(* IEC 61131-3 sources: SmartHomeNew/snapshots/2026-05-19 (part 3) *)

(* ---- FB_Heating_Runtime_Timeline_Observer.st ---- *)
// ==============================================================================
// Heating runtime timeline observer
// Read-only deterministic execution timeline layer.
// ==============================================================================
FUNCTION_BLOCK FB_Heating_Runtime_Timeline_Observer
VAR_INPUT
    VI_Enable : BOOL;
    VI_Frame : ST_Heating_Runtime_Execution_Frame;
END_VAR
VAR_IN_OUT
    VIO_Timeline : ST_Heating_Runtime_Execution_Timeline;
END_VAR
VAR
    L_Index : UINT;
END_VAR

IF NOT VI_Enable THEN
    RETURN;
END_IF;

// ======================================================
// SAFE INDEX NORMALIZATION
// ======================================================
IF (VIO_Timeline.Write_Index < 1) OR
   (VIO_Timeline.Write_Index >= 64) THEN

    L_Index := 1;

    IF VIO_Timeline.Write_Index >= 64 THEN
        VIO_Timeline.Timeline_Overflow := TRUE;
    END_IF;

ELSE
    L_Index := VIO_Timeline.Write_Index + 1;
END_IF;

// ======================================================
// FRAME STORAGE
// ======================================================
VIO_Timeline.Frames[L_Index] := VI_Frame;
VIO_Timeline.Write_Index := L_Index;

IF VIO_Timeline.Frame_Count < 64 THEN
    VIO_Timeline.Frame_Count :=
        VIO_Timeline.Frame_Count + 1;
END_IF;

// ======================================================
// TELEMETRY UPDATE
// ======================================================
VIO_Timeline.Sequencing_Valid :=
    VI_Frame.Sequencing_Valid;

VIO_Timeline.Ownership_Valid :=
    VI_Frame.Ownership_Valid;

VIO_Timeline.Synchronization_Valid :=
    VI_Frame.Synchronization_Valid;

VIO_Timeline.Runtime_Jitter_Detected :=
    VI_Frame.Runtime_Jitter_Detected;

VIO_Timeline.Runtime_Latency_Detected :=
    VI_Frame.Runtime_Latency_Detected;

VIO_Timeline.Runtime_Degraded :=
    VI_Frame.Runtime_Degraded;

VIO_Timeline.Status_Code := VI_Frame.Status_Code;
VIO_Timeline.Status_Text := VI_Frame.Status_Text;

END_FUNCTION_BLOCK
// >>> BULK_SYNC_ANCHOR: FB_Heating_Runtime_Timeline_Observer <<<

(* ---- FB_Heating_Safe_State.st ---- *)
FUNCTION_BLOCK FB_Heating_Safe_State
VAR_INPUT
    VI_Block_Normal_Heating : BOOL;
    VI_IO_Failsafe_Active : BOOL;
    VI_Gas_Safety_Active : BOOL;
    VI_Freeze_Active : BOOL;
    VI_Freeze_Target_Supply : REAL;
    VI_Manifold_Temps_Supply : ARRAY[1..GVL_CONSTANTS.C_MAX_MANIFOLDS] OF REAL;
    VI_Boiler_Error_Status : ARRAY[1..GVL_CONSTANTS.C_MAX_BOILERS] OF BOOL;
    VI_Boiler_OT_Online : ARRAY[1..GVL_CONSTANTS.C_MAX_BOILERS] OF BOOL;
END_VAR
VAR_OUTPUT
    VO_Applied : BOOL;
    VO_Zone_Valves : ARRAY[1..GVL_CONSTANTS.C_MAX_HEATING_CIRCUITS] OF BOOL;
    VO_Manifold_Pumps : ARRAY[1..GVL_CONSTANTS.C_MAX_MANIFOLDS] OF BOOL;
    VO_Manifold_Valves : ARRAY[1..GVL_CONSTANTS.C_MAX_MANIFOLDS] OF REAL;
    VO_Boiler_OT_Enable : ARRAY[1..GVL_CONSTANTS.C_MAX_BOILERS] OF BOOL;
    VO_Boiler_OT_Setpoint : ARRAY[1..GVL_CONSTANTS.C_MAX_BOILERS] OF REAL;
    VO_Boiler_Status : ARRAY[1..GVL_CONSTANTS.C_MAX_BOILERS] OF ST_Boiler_Status;
    VO_Backup_Circulation_Pump : BOOL;
    VO_Electric_Heater_Enable : BOOL;
    VO_Freeze_Risk_Status : BOOL;
END_VAR
VAR
    L_i : INT;
    L_Min_Supply_Temp : REAL;
    L_Freeze_Circulation_Required : BOOL;
END_VAR

VO_Applied := VI_Block_Normal_Heating;
VO_Backup_Circulation_Pump := FALSE;
VO_Electric_Heater_Enable := FALSE;
VO_Freeze_Risk_Status := FALSE;

L_Freeze_Circulation_Required := VI_Freeze_Active AND (VI_IO_Failsafe_Active OR VI_Gas_Safety_Active);

IF NOT VI_Block_Normal_Heating THEN
    RETURN;
END_IF;

// =============================
// ZONE VALVES (FIXED)
// =============================
FOR L_i := 1 TO GVL_CONSTANTS.C_MAX_HEATING_CIRCUITS DO
    IF L_Freeze_Circulation_Required THEN
        VO_Zone_Valves[L_i] := TRUE;
    ELSE
        VO_Zone_Valves[L_i] := FALSE;
    END_IF;
END_FOR;

// =============================
// MANIFOLD CONTROL
// =============================
FOR L_i := 1 TO GVL_CONSTANTS.C_MAX_MANIFOLDS DO
    IF L_Freeze_Circulation_Required THEN
        VO_Manifold_Pumps[L_i] := TRUE;
        VO_Manifold_Valves[L_i] := REAL#35.0;
    ELSE
        VO_Manifold_Pumps[L_i] := FALSE;
        VO_Manifold_Valves[L_i] := REAL#0.0;
    END_IF;
END_FOR;

// =============================
// BOILERS OFF
// =============================
FOR L_i := 1 TO GVL_CONSTANTS.C_MAX_BOILERS DO
    VO_Boiler_OT_Enable[L_i] := FALSE;
    VO_Boiler_OT_Setpoint[L_i] := REAL#0.0;
    VO_Boiler_Status[L_i].Warning := FALSE;
    VO_Boiler_Status[L_i].Error := TRUE;
END_FOR;

// =============================
// FREEZE PROTECTION LOGIC
// =============================
IF VI_Gas_Safety_Active AND VI_Freeze_Active THEN
    VO_Backup_Circulation_Pump := TRUE;

    L_Min_Supply_Temp := REAL#1000.0;
    FOR L_i := 1 TO GVL_CONSTANTS.C_MAX_MANIFOLDS DO
        IF VI_Manifold_Temps_Supply[L_i] < L_Min_Supply_Temp THEN
            L_Min_Supply_Temp := VI_Manifold_Temps_Supply[L_i];
        END_IF;
    END_FOR;

    IF L_Min_Supply_Temp > REAL#900.0 THEN
        L_Min_Supply_Temp := REAL#0.0;
    END_IF;

    IF L_Min_Supply_Temp < (VI_Freeze_Target_Supply - REAL#1.0) THEN
        VO_Electric_Heater_Enable := TRUE;
    ELSIF L_Min_Supply_Temp > (VI_Freeze_Target_Supply + REAL#1.0) THEN
        VO_Electric_Heater_Enable := FALSE;
    END_IF;

    VO_Freeze_Risk_Status := TRUE;
END_IF;

// =============================
// IO FAILSAFE + FREEZE
// =============================
IF VI_IO_Failsafe_Active AND VI_Freeze_Active THEN
    IF VI_Boiler_OT_Online[1] AND NOT VI_Boiler_Error_Status[1] THEN
        VO_Boiler_OT_Enable[1] := TRUE;
        VO_Boiler_OT_Setpoint[1] := VI_Freeze_Target_Supply;
    END_IF;
END_IF;

END_FUNCTION_BLOCK
// >>> BULK_SYNC_ANCHOR: FB_Heating_Safe_State <<<

(* ---- FB_Heating_System_Manager.st ---- *)
FUNCTION_BLOCK FB_Heating_System_Manager
VAR_INPUT
    VI_System_Mode : E_System_Operating_Mode;
    VI_System_Time_MS : UDINT;
    VI_IsActivePLC : BOOL;
    VI_Outdoor_Temp : REAL;
    VI_Config : ST_Heating_Config;
    VI_Tariff : ST_Tariff_Config;
    VI_Current_Hour : UINT;
    VI_DHW_Heating_Demand : BOOL;
    VI_DHW_Target_Temp : REAL;
    VI_Emergency_Stop : BOOL;
    VI_Gas_Safety_Stop : BOOL;
    VI_Boiler_Error_Status : ARRAY[1..GVL_CONSTANTS.C_MAX_BOILERS] OF BOOL;
    VI_Boiler_OT_Online : ARRAY[1..GVL_CONSTANTS.C_MAX_BOILERS] OF BOOL;
    VI_Boiler_Modulation : ARRAY[1..GVL_CONSTANTS.C_MAX_BOILERS] OF REAL;
END_VAR
VAR_IN_OUT
    VI_Floor_Temps : ARRAY[1..GVL_CONSTANTS.C_MAX_HEATING_CIRCUITS] OF REAL;
    VI_Room_Temps : ARRAY[1..GVL_CONSTANTS.C_MAX_ZONES] OF REAL;
    VI_Manifold_Pressures : ARRAY[1..GVL_CONSTANTS.C_MAX_MANIFOLDS] OF REAL;
    VI_Manifold_Currents : ARRAY[1..GVL_CONSTANTS.C_MAX_MANIFOLDS] OF REAL;
    VI_Manifold_Temps_Supply : ARRAY[1..GVL_CONSTANTS.C_MAX_MANIFOLDS] OF REAL;
    VI_Manifold_Temps_Return : ARRAY[1..GVL_CONSTANTS.C_MAX_MANIFOLDS] OF REAL;
    VI_Boiler_Flame_Status : ARRAY[1..GVL_CONSTANTS.C_MAX_BOILERS] OF BOOL;
    VI_Zone_Configs : ARRAY[1..GVL_CONSTANTS.C_MAX_HEATING_CIRCUITS] OF ST_FloorHeating_Circuit_Config;
    VI_Rule_Actions : ARRAY[1..GVL_CONSTANTS.C_MAX_RULES] OF ST_Rule_Action;
    VI_IO_Modules_Online : ARRAY[1..GVL_CONSTANTS.C_MAX_MODULES] OF BOOL;
    VI_Manifold_End_Switches : ARRAY[1..GVL_CONSTANTS.C_MAX_MANIFOLDS] OF BOOL;
    VI_Valve_Test_Config : ARRAY[1..GVL_CONSTANTS.C_MAX_MANIFOLDS] OF ST_Valve_Test_Config;
END_VAR
VAR_OUTPUT
    VO_Manifold_Valves : ARRAY[1..GVL_CONSTANTS.C_MAX_MANIFOLDS] OF REAL;
    VO_Manifold_Pumps : ARRAY[1..GVL_CONSTANTS.C_MAX_MANIFOLDS] OF BOOL;
    VO_Zone_Valves : ARRAY[1..GVL_CONSTANTS.C_MAX_HEATING_CIRCUITS] OF BOOL;
    VO_Boiler_OT_Enable : ARRAY[1..GVL_CONSTANTS.C_MAX_BOILERS] OF BOOL;
    VO_Boiler_OT_Setpoint : ARRAY[1..GVL_CONSTANTS.C_MAX_BOILERS] OF REAL;
    VO_Backup_Circulation_Pump : BOOL;
    VO_Electric_Heater_Enable : BOOL;
    VO_Freeze_Risk_Status : BOOL;
    VO_Status : ARRAY[1..GVL_CONSTANTS.C_MAX_MANIFOLDS] OF ST_Manifold_Status;
    VO_Boiler_Status : ARRAY[1..GVL_CONSTANTS.C_MAX_BOILERS] OF ST_Boiler_Status;
END_VAR
VAR
    L_i : INT;
    L_Target_Supply_Temp : REAL;
    L_Manifold_Demand_Map : ARRAY[1..GVL_CONSTANTS.C_MAX_MANIFOLDS] OF BOOL;
    L_Manifold_Demand_Filtered : ARRAY[1..GVL_CONSTANTS.C_MAX_MANIFOLDS] OF BOOL;
    L_Manifold_Available : ARRAY[1..GVL_CONSTANTS.C_MAX_MANIFOLDS] OF BOOL;
    L_Manifold_In_Service : ARRAY[1..GVL_CONSTANTS.C_MAX_MANIFOLDS] OF BOOL;
    L_Manifold_Subsystem_Degraded : ARRAY[1..GVL_CONSTANTS.C_MAX_MANIFOLDS] OF BOOL;
    L_Manifold_Base_Priority : ARRAY[1..GVL_CONSTANTS.C_MAX_MANIFOLDS] OF INT;
    L_Manifold_Effective_Priority : ARRAY[1..GVL_CONSTANTS.C_MAX_MANIFOLDS] OF INT;
    L_Manifold_Thermal_Weight : ARRAY[1..GVL_CONSTANTS.C_MAX_MANIFOLDS] OF REAL;
    L_Allocation_Degraded : BOOL;
    fbValveTestManager : FB_Valve_Test_Manager;
    L_IO_Failsafe_Active : BOOL;
    L_Freeze_Active : BOOL;
    L_Freeze_Target_Supply : REAL;
    L_Policy_Degraded : BOOL;
    L_Sensor_Error : BOOL;
    L_Subsys_Degraded : BOOL;
    L_Pressure_OK : BOOL;
    L_Prev_Pressure : ARRAY[1..GVL_CONSTANTS.C_MAX_MANIFOLDS] OF REAL;
    L_Prev_Current : ARRAY[1..GVL_CONSTANTS.C_MAX_MANIFOLDS] OF REAL;
    L_Confidence : REAL;
    L_Policy_Target_Adjustment : REAL;
    fbAdaptiveTarget : FB_Heating_Adaptive_Target;
    fbSafetyGate : FB_Heating_Safety_Gate;
    fbSafeState : FB_Heating_Safe_State;
    fbDemandMap : FB_Heating_Demand_Map;
    fbPolicyPriorityBridge : FB_Heating_Policy_Priority_Bridge;
    fbAllocationFilter : FB_Heating_Allocation_Filter;
    fbRuntimeObservability : FB_Heating_Runtime_Observability;
    fbCircuitControl : FB_Heating_Circuit_Control;
    fbManifoldControl : FB_Heating_Manifold_Control;
    fbBoilerControl : FB_Heating_Boiler_Control;
END_VAR

L_Policy_Degraded := (VI_System_Mode = E_System_Operating_Mode.MODE_DEGRADED);

GVL_STATE.G_Heating_IO_Fault := FALSE;
GVL_STATE.G_Heating_Sensor_Fault := FALSE;
GVL_STATE.G_Heating_Subsystem_Degraded := FALSE;
L_Sensor_Error := FALSE;
L_Subsys_Degraded := FALSE;
L_Allocation_Degraded := FALSE;

L_IO_Failsafe_Active := FALSE;
FOR L_i := 1 TO GVL_CONSTANTS.C_MAX_MODULES DO
    IF NOT VI_IO_Modules_Online[L_i] THEN
        L_IO_Failsafe_Active := TRUE;
        GVL_STATE.G_Heating_IO_Fault := TRUE;
        GVL_STATE.G_Heating_Subsystem_Degraded := TRUE;
        EXIT;
    END_IF;
END_FOR;

fbSafetyGate(
    VI_System_Mode := VI_System_Mode,
    VI_Emergency_Stop := VI_Emergency_Stop,
    VI_Gas_Safety_Stop := VI_Gas_Safety_Stop,
    VI_IO_Failsafe_Active := L_IO_Failsafe_Active,
    VI_Outdoor_Temp := VI_Outdoor_Temp,
    VI_Freeze_Threshold := VI_Config.Freeze_Threshold,
    VI_Floor_Temps := VI_Floor_Temps,
    VO_Freeze_Mode_Active => L_Freeze_Active,
    VO_Freeze_Target_Supply => L_Freeze_Target_Supply
);

fbSafeState(
    VI_Block_Normal_Heating := fbSafetyGate.VO_Block_Normal_Heating,
    VI_IO_Failsafe_Active := fbSafetyGate.VO_IO_Failsafe_Active,
    VI_Gas_Safety_Active := fbSafetyGate.VO_Gas_Safety_Active,
    VI_Freeze_Active := L_Freeze_Active,
    VI_Freeze_Target_Supply := L_Freeze_Target_Supply,
    VI_Manifold_Temps_Supply := VI_Manifold_Temps_Supply,
    VI_Boiler_Error_Status := VI_Boiler_Error_Status,
    VI_Boiler_OT_Online := VI_Boiler_OT_Online
);

IF fbSafeState.VO_Applied THEN
    FOR L_i := 1 TO GVL_CONSTANTS.C_MAX_HEATING_CIRCUITS DO
        VO_Zone_Valves[L_i] := fbSafeState.VO_Zone_Valves[L_i];
    END_FOR;

    FOR L_i := 1 TO GVL_CONSTANTS.C_MAX_MANIFOLDS DO
        VO_Manifold_Pumps[L_i] := fbSafeState.VO_Manifold_Pumps[L_i];
        VO_Manifold_Valves[L_i] := fbSafeState.VO_Manifold_Valves[L_i];
    END_FOR;

    FOR L_i := 1 TO GVL_CONSTANTS.C_MAX_BOILERS DO
        VO_Boiler_OT_Enable[L_i] := fbSafeState.VO_Boiler_OT_Enable[L_i];
        VO_Boiler_OT_Setpoint[L_i] := fbSafeState.VO_Boiler_OT_Setpoint[L_i];
        VO_Boiler_Status[L_i] := fbSafeState.VO_Boiler_Status[L_i];
    END_FOR;

    VO_Backup_Circulation_Pump := fbSafeState.VO_Backup_Circulation_Pump;
    VO_Electric_Heater_Enable := fbSafeState.VO_Electric_Heater_Enable;
    VO_Freeze_Risk_Status := fbSafeState.VO_Freeze_Risk_Status;
    RETURN;
END_IF;

VO_Backup_Circulation_Pump := FALSE;
VO_Electric_Heater_Enable := FALSE;
VO_Freeze_Risk_Status := FALSE;

IF L_Freeze_Active THEN
    L_Target_Supply_Temp := L_Freeze_Target_Supply;
ELSE
    L_Target_Supply_Temp := VI_Config.Target_Floor_Temp;
END_IF;

fbAdaptiveTarget(
    VI_Base_Target_Supply_Temp := L_Target_Supply_Temp,
    VI_Global_Target_Temperature := GVL_STATE.G_Target_Temperature,
    VI_Zone_Configs := VI_Zone_Configs,
    VI_Floor_Temps := VI_Floor_Temps,
    VI_Room_Temps := VI_Room_Temps,
    VO_Target_Supply_Temp => L_Target_Supply_Temp
);

L_Policy_Target_Adjustment := GVL_HEATING_POLICY.G_Policy_Target_Adjustment;

IF L_Policy_Target_Adjustment > REAL#5.0 THEN
    L_Policy_Target_Adjustment := REAL#5.0;
ELSIF L_Policy_Target_Adjustment < REAL#-3.0 THEN
    L_Policy_Target_Adjustment := REAL#-3.0;
END_IF;

L_Target_Supply_Temp :=
    LIMIT(
        GVL_CONSTANTS.C_BOILER_SETPOINT_MIN,
        L_Target_Supply_Temp + L_Policy_Target_Adjustment,
        GVL_CONSTANTS.C_BOILER_SETPOINT_MAX
    );

fbCircuitControl(
    VI_System_Time_MS := VI_System_Time_MS,
    VI_Current_Hour := VI_Current_Hour,
    VI_IsActivePLC := VI_IsActivePLC,
    VI_Config := VI_Config,
    VI_Tariff := VI_Tariff,
    VI_Scenario_Adjust := REAL#0.0,
    VI_Zone_Configs := VI_Zone_Configs,
    VI_Floor_Temps := VI_Floor_Temps,
    VI_Room_Temps := VI_Room_Temps,
    VI_Rule_Actions := VI_Rule_Actions,
    VO_Zone_Valves => VO_Zone_Valves,
    VO_Heating_Sensor_Fault => L_Sensor_Error
);

GVL_STATE.G_Heating_Sensor_Fault := L_Sensor_Error;

fbDemandMap(
    VI_Zone_Valves := VO_Zone_Valves,
    VI_Zone_Configs := VI_Zone_Configs,
    VO_Manifold_Demand_Map => L_Manifold_Demand_Map
);

FOR L_i := 1 TO GVL_CONSTANTS.C_MAX_MANIFOLDS DO
    L_Manifold_Available[L_i] := VI_Manifold_Pressures[L_i] >= GVL_CONSTANTS.C_MIN_HEATING_MANIFOLD_PRESSURE;
    L_Manifold_In_Service[L_i] := GVL_CONFIG.G_Manifold_Pump_In_Service[L_i];
    L_Manifold_Subsystem_Degraded[L_i] :=
        GVL_STATE.G_Predictive_Pump_Pressure_Drop[L_i]
        OR GVL_STATE.G_Predictive_Pump_Current_Rise[L_i];

    L_Manifold_Base_Priority[L_i] := GVL_CONFIG.G_Manifold_Priority[L_i];
    L_Manifold_Thermal_Weight[L_i] := GVL_CONFIG.G_Manifold_Thermal_Weight[L_i];
END_FOR;

fbPolicyPriorityBridge(
    VI_Enable := (GVL_CONFIG.G_Max_Thermal_Budget > REAL#0.0),
    VI_Zone_Valves := VO_Zone_Valves,
    VI_Zone_Configs := VI_Zone_Configs,
    VI_Manifold_Base_Priority := L_Manifold_Base_Priority,
    VI_Zone_Priority_Bias := GVL_HEATING_POLICY.G_Zone_Priority_Bias,
    VI_Policy_Priority_Multiplier := GVL_HEATING_POLICY.G_Policy_Priority_Multiplier,
    VO_Manifold_Effective_Priority => L_Manifold_Effective_Priority
);

fbAllocationFilter(
    VI_Enable := TRUE,
    VI_Enable_Policy_Allocation := (GVL_CONFIG.G_Max_Thermal_Budget > REAL#0.0),
    VI_Freeze_Mode_Active := L_Freeze_Active,
    VI_DHW_Heating_Demand := VI_DHW_Heating_Demand,
    VI_Manifold_Demand_Map := L_Manifold_Demand_Map,
    VI_Manifold_Available := L_Manifold_Available,
    VI_Manifold_In_Service := L_Manifold_In_Service,
    VI_Manifold_Subsystem_Degraded := L_Manifold_Subsystem_Degraded,
    VI_Manifold_Base_Priority := L_Manifold_Effective_Priority,
    VI_Manifold_Thermal_Weight := L_Manifold_Thermal_Weight,
    VI_Max_Thermal_Budget := GVL_CONFIG.G_Max_Thermal_Budget,
    VO_Manifold_Demand_Filtered => L_Manifold_Demand_Filtered,
    VO_Allocation_Degraded => L_Allocation_Degraded
);

fbRuntimeObservability(
    VI_Policy_Active := (GVL_CONFIG.G_Max_Thermal_Budget > REAL#0.0),
    VI_Freeze_Bypass_Active := L_Freeze_Active,
    VI_DHW_Bypass_Active := VI_DHW_Heating_Demand,
    VI_Budget_Max := GVL_CONFIG.G_Max_Thermal_Budget,
    VI_Budget_Used := fbAllocationFilter.VO_Thermal_Budget_Used,
    VI_Requested := L_Manifold_Demand_Map,
    VI_Allowed := fbAllocationFilter.VO_Manifold_Allowed,
    VI_Filtered := L_Manifold_Demand_Filtered,
    VI_Block_Reason := fbAllocationFilter.VO_Manifold_Block_Reason,
    VI_Effective_Priority := fbAllocationFilter.VO_Manifold_Priority_Effective,
    VI_Priority_Bridge_Active := fbPolicyPriorityBridge.VO_Bridge_Active,
    VI_Priority_Bias_Applied := fbPolicyPriorityBridge.VO_Manifold_Priority_Bias_Applied,
    VI_Priority_Effective := L_Manifold_Effective_Priority
);

IF L_Allocation_Degraded THEN
    GVL_STATE.G_Heating_Subsystem_Degraded := TRUE;
END_IF;

fbManifoldControl(
    VI_System_Time_MS := VI_System_Time_MS,
    VI_IsActivePLC := VI_IsActivePLC,
    VI_DHW_Heating_Demand := VI_DHW_Heating_Demand,
    VI_Freeze_Mode_Active := L_Freeze_Active,
    VI_Target_Supply_Temp := L_Target_Supply_Temp,
    VI_Any_Zone_Active := L_Manifold_Demand_Filtered,
    VI_Manifold_Pressures := VI_Manifold_Pressures,
    VI_Manifold_Currents := VI_Manifold_Currents,
    VI_Manifold_Temps_Supply := VI_Manifold_Temps_Supply,
    VI_Manifold_Temps_Return := VI_Manifold_Temps_Return,
    VO_Manifold_Pumps => VO_Manifold_Pumps,
    VO_Manifold_Valves => VO_Manifold_Valves,
    VO_Status => VO_Status
);

FOR L_i := 1 TO GVL_CONSTANTS.C_MAX_MANIFOLDS DO
    L_Pressure_OK := VI_Manifold_Pressures[L_i] >= GVL_CONSTANTS.C_MIN_HEATING_MANIFOLD_PRESSURE;

    IF VO_Manifold_Pumps[L_i] AND NOT L_Pressure_OK THEN
        VO_Manifold_Pumps[L_i] := FALSE;
        GVL_STATE.G_Heating_Subsystem_Degraded := TRUE;
    END_IF;

    IF (L_Prev_Pressure[L_i] > REAL#0.0) AND ((L_Prev_Pressure[L_i] - VI_Manifold_Pressures[L_i]) > REAL#0.2) THEN
        GVL_STATE.G_Predictive_Pump_Pressure_Drop[L_i] := TRUE;
    ELSE
        GVL_STATE.G_Predictive_Pump_Pressure_Drop[L_i] := FALSE;
    END_IF;

    IF (L_Prev_Current[L_i] > REAL#0.0) AND (VI_Manifold_Currents[L_i] > (L_Prev_Current[L_i] * REAL#1.2)) THEN
        GVL_STATE.G_Predictive_Pump_Current_Rise[L_i] := TRUE;
    ELSE
        GVL_STATE.G_Predictive_Pump_Current_Rise[L_i] := FALSE;
    END_IF;

    IF GVL_STATE.G_Predictive_Pump_Pressure_Drop[L_i] OR GVL_STATE.G_Predictive_Pump_Current_Rise[L_i] THEN
        GVL_STATE.G_Heating_Subsystem_Degraded := TRUE;
    END_IF;

    L_Prev_Pressure[L_i] := VI_Manifold_Pressures[L_i];
    L_Prev_Current[L_i] := VI_Manifold_Currents[L_i];
END_FOR;

// ======================================================
// HEATING CONFIDENCE PUBLICATION
// ======================================================
// The former local error-score decay path has been replaced by the
// normalized input confidence surface. Runtime faults may still reduce
// confidence and reason publication, but the base confidence now comes
// from canonical input semantics.
L_Confidence := GVL_INPUT.IN_Min_Zone_Confidence;

IF L_Confidence < REAL#0.0 THEN
    L_Confidence := REAL#0.0;
ELSIF L_Confidence > REAL#1.0 THEN
    L_Confidence := REAL#1.0;
END_IF;

GVL_STATE.G_Heating_Confidence_Reason_Code := 0;
GVL_STATE.G_Heating_Confidence_Reason_Text := 'OK';

IF GVL_INPUT.IN_Input_Degraded OR GVL_INPUT.IN_Anomaly_Detected THEN
    GVL_STATE.G_Heating_Subsystem_Degraded := TRUE;
    GVL_STATE.G_Heating_Confidence_Reason_Code := 5;

    IF GVL_INPUT.IN_Anomaly_Reason <> '' THEN
        GVL_STATE.G_Heating_Confidence_Reason_Text := GVL_INPUT.IN_Anomaly_Reason;
    ELSE
        GVL_STATE.G_Heating_Confidence_Reason_Text := 'Input quality degraded';
    END_IF;
END_IF;

IF GVL_STATE.G_Heating_IO_Fault THEN
    IF L_Confidence > REAL#0.8 THEN
        L_Confidence := REAL#0.8;
    END_IF;
    GVL_STATE.G_Heating_Confidence_Reason_Code := 2;
    GVL_STATE.G_Heating_Confidence_Reason_Text := 'IO fault detected';
ELSIF GVL_STATE.G_Heating_Sensor_Fault THEN
    IF L_Confidence > REAL#0.6 THEN
        L_Confidence := REAL#0.6;
    END_IF;
    GVL_STATE.G_Heating_Confidence_Reason_Code := 1;
    GVL_STATE.G_Heating_Confidence_Reason_Text := 'Sensor fault detected';
ELSE
    FOR L_i := 1 TO GVL_CONSTANTS.C_MAX_MANIFOLDS DO
        IF VI_Manifold_Pressures[L_i] < GVL_CONSTANTS.C_MIN_HEATING_MANIFOLD_PRESSURE THEN
            IF L_Confidence > REAL#0.7 THEN
                L_Confidence := REAL#0.7;
            END_IF;
            GVL_STATE.G_Heating_Confidence_Reason_Code := 3;
            GVL_STATE.G_Heating_Confidence_Reason_Text := 'Low manifold pressure';
            EXIT;
        END_IF;
    END_FOR;

    FOR L_i := 1 TO GVL_CONSTANTS.C_MAX_MANIFOLDS DO
        IF GVL_STATE.G_Predictive_Pump_Pressure_Drop[L_i] OR GVL_STATE.G_Predictive_Pump_Current_Rise[L_i] THEN
            IF L_Confidence > REAL#0.75 THEN
                L_Confidence := REAL#0.75;
            END_IF;
            GVL_STATE.G_Heating_Confidence_Reason_Code := 4;
            GVL_STATE.G_Heating_Confidence_Reason_Text := 'Predictive pump degradation';
            EXIT;
        END_IF;
    END_FOR;
END_IF;

GVL_STATE.G_Heating_Confidence := L_Confidence;
GVL_STATE.G_Heating_Error_Score := REAL#1.0 - L_Confidence;

IF GVL_STATE.G_Heating_Confidence < REAL#0.5 THEN
    L_Target_Supply_Temp := L_Target_Supply_Temp - REAL#3.0;
END_IF;

CASE GVL_STATE.G_Heating_Confidence_Reason_Code OF
    1:
        L_Target_Supply_Temp := LIMIT(GVL_CONSTANTS.C_BOILER_SETPOINT_MIN, REAL#40.0, GVL_CONSTANTS.C_BOILER_SETPOINT_MAX);
    2:
        VO_Backup_Circulation_Pump := TRUE;
    3:
        FOR L_i := 1 TO GVL_CONSTANTS.C_MAX_MANIFOLDS DO
            VO_Manifold_Pumps[L_i] := FALSE;
        END_FOR;
    4:
        L_Target_Supply_Temp := LIMIT(GVL_CONSTANTS.C_BOILER_SETPOINT_MIN, L_Target_Supply_Temp - REAL#5.0, GVL_CONSTANTS.C_BOILER_SETPOINT_MAX);
    5:
        // Input-quality degradation is published for explainability first.
        // Runtime suppression remains governed by existing sensor validation
        // and safety/pressure ownership paths.
ELSE
    // no auto-recovery action
END_CASE;

fbValveTestManager(
    VI_System_Time_MS := VI_System_Time_MS,
    VI_IsActivePLC := VI_IsActivePLC,
    VI_Valve_Currents := VI_Manifold_Currents,
    VI_Valve_End_Switches := VI_Manifold_End_Switches,
    VI_Config := VI_Valve_Test_Config
);

IF fbValveTestManager.VO_Test_Active THEN
    L_i := fbValveTestManager.VO_Current_Valve;
    IF L_i >= 1 AND L_i <= GVL_CONSTANTS.C_MAX_MANIFOLDS THEN
        IF fbValveTestManager.VO_Valve_Cmd[L_i] THEN
            VO_Manifold_Valves[L_i] := REAL#100.0;
        ELSE
            VO_Manifold_Valves[L_i] := REAL#0.0;
        END_IF;
        VO_Manifold_Pumps[L_i] := FALSE;
    END_IF;
END_IF;

fbBoilerControl(
    VI_System_Time_MS := VI_System_Time_MS,
    VI_IsActivePLC := VI_IsActivePLC,
    VI_DHW_Heating_Demand := VI_DHW_Heating_Demand,
    VI_DHW_Target_Temp := VI_DHW_Target_Temp,
    VI_Target_Supply_Temp := L_Target_Supply_Temp,
    VI_Freeze_Mode_Active := L_Freeze_Active,
    VI_Policy_Degraded := L_Policy_Degraded,
    VI_Manifold_Pumps := VO_Manifold_Pumps,
    VI_Manifold_Valves := VO_Manifold_Valves,
    VI_Boiler_Flame_Status := VI_Boiler_Flame_Status,
    VI_Boiler_Error_Status := VI_Boiler_Error_Status,
    VI_Boiler_OT_Online := VI_Boiler_OT_Online,
    VI_Boiler_Modulation := VI_Boiler_Modulation,
    VO_Boiler_OT_Enable => VO_Boiler_OT_Enable,
    VO_Boiler_OT_Setpoint => VO_Boiler_OT_Setpoint,
    VO_Boiler_Status => VO_Boiler_Status,
    VO_Any_Subsystem_Degraded => L_Subsys_Degraded
);

GVL_STATE.G_Heating_Subsystem_Degraded := GVL_STATE.G_Heating_Subsystem_Degraded OR L_Subsys_Degraded;

END_FUNCTION_BLOCK
// >>> BULK_SYNC_ANCHOR: FB_Heating_System_Manager <<<

(* ---- FB_History_Manager.st ---- *)
FUNCTION_BLOCK FB_History_Manager
VAR_INPUT
    VI_System_Time_MS : UDINT;
    VI_Write_Event    : BOOL;
    VI_Event          : ST_History_Record;
END_VAR
VAR_OUTPUT
    VO_Total_Events   : UDINT;
END_VAR
VAR
    L_Prev_Write_Event : BOOL;
END_VAR

IF VI_Write_Event AND NOT L_Prev_Write_Event THEN
    GVL_Retain.G_History_Buffer[GVL_Retain.G_History_Write_Idx] := VI_Event;
    GVL_Retain.G_History_Buffer[GVL_Retain.G_History_Write_Idx].timestamp_ms := VI_System_Time_MS;

    GVL_Retain.G_History_Write_Idx := (GVL_Retain.G_History_Write_Idx MOD GVL_CONSTANTS.C_MAX_HISTORY_RECORDS) + 1;
    GVL_Retain.G_History_Total_Events := GVL_Retain.G_History_Total_Events + 1;
END_IF;
L_Prev_Write_Event := VI_Write_Event;

VO_Total_Events := GVL_Retain.G_History_Total_Events;
// >>> BULK_SYNC_ANCHOR: FB_History_Manager <<<
END_FUNCTION_BLOCK

(* ---- FB_HMI_Config_Workflow_Runtime.st ---- *)
FUNCTION_BLOCK FB_HMI_Config_Workflow_Runtime
VAR_INPUT
    VI_Enable : BOOL;
    VI_System_Time_MS : UDINT;
END_VAR
VAR
    L_State : ST_HMI_Config_Workflow_State;
END_VAR

IF NOT VI_Enable THEN
    GVL_HMI_Config_Workflow.G_Runtime_Valid := FALSE;
    RETURN;
END_IF;

L_State.Runtime_Valid := TRUE;
L_State.Runtime_System_Time_MS := VI_System_Time_MS;

L_State.Editor_Open :=
    GVL_HMI_Config_Workflow.G_Open_Editor_Request;

L_State.Validation_Requested :=
    GVL_HMI_Config_Workflow.G_Validate_Request;

L_State.Activation_Requested :=
    GVL_HMI_Config_Workflow.G_Activate_Request;

L_State.Rollback_Requested :=
    GVL_HMI_Config_Workflow.G_Rollback_Request;

L_State.Active_Version :=
    GVL_Water_Topology_Config.G_Active_Config_Version;

L_State.Draft_Version :=
    GVL_Config_Activation.G_Staged_Config_Version;

L_State.Last_Stable_Version :=
    GVL_Config_Activation.G_Last_Stable_Config_Version;

L_State.Quarantine_Visible :=
    GVL_Config_Activation.G_Config_Quarantine_Active;

L_State.Service_Mode_Required := TRUE;
L_State.Operator_Ack_Required := TRUE;

IF L_State.Editor_Open THEN
    L_State.Edit_Session_Active := TRUE;
END_IF;

IF L_State.Validation_Requested THEN

    IF GVL_Config_Activation.G_Activation_State.Staged_Config_Valid THEN

        L_State.Validation_OK := TRUE;

    ELSE

        L_State.Validation_Failed := TRUE;

    END_IF;

END_IF;

IF L_State.Activation_Requested THEN

    IF GVL_HMI_Config_Workflow.G_Service_Mode_Active
       AND GVL_HMI_Config_Workflow.G_Operator_Ack
       AND L_State.Validation_OK THEN

        L_State.Activation_Allowed := TRUE;
        GVL_Config_Activation.G_Activation_Request := TRUE;

    ELSE

        L_State.Activation_Blocked := TRUE;

    END_IF;

END_IF;

IF L_State.Rollback_Requested THEN

    IF GVL_HMI_Config_Workflow.G_Operator_Ack THEN

        L_State.Rollback_Allowed := TRUE;
        GVL_Config_Activation.G_Rollback_Request := TRUE;

    END_IF;

END_IF;

IF L_State.Activation_Blocked THEN

    L_State.Status_Code := 2;
    L_State.Status_Text := 'HMI activation blocked';

ELSIF L_State.Validation_Failed THEN

    L_State.Status_Code := 1;
    L_State.Status_Text := 'HMI validation failed';

ELSE

    L_State.Status_Code := 0;
    L_State.Status_Text := 'HMI config workflow healthy';

END_IF;

GVL_HMI_Config_Workflow.G_Workflow_State := L_State;

GVL_HMI_Config_Workflow.G_Runtime_Valid := TRUE;
GVL_HMI_Config_Workflow.G_Last_Update_MS := VI_System_Time_MS;
GVL_HMI_Config_Workflow.G_Status_Code := L_State.Status_Code;
GVL_HMI_Config_Workflow.G_Status_Text := L_State.Status_Text;

END_FUNCTION_BLOCK

(* ---- FB_IO_Module_Watchdog.st ---- *)
FUNCTION_BLOCK FB_IO_Module_Watchdog
VAR_INPUT
    VI_System_Time_MS : UDINT;
    VI_Module_ID : BYTE;
    VI_Heartbeat_Signal : BOOL; // Сигнал от модуля (например, мигающий бит)
    VI_Timeout_MS : UDINT := 2000; // Таймаут 2 секунды по умолчанию
END_VAR
VAR_OUTPUT
    VO_Module_Online : BOOL;
    VO_Error_Active : BOOL;
END_VAR
VAR
    L_Last_Heartbeat_State : BOOL;
    L_Last_Heartbeat_Time : UDINT;
    L_Elapsed_Time : UDINT;
END_VAR

// Отслеживание изменения сигнала
IF VI_Heartbeat_Signal <> L_Last_Heartbeat_State THEN
    L_Last_Heartbeat_Time := VI_System_Time_MS;
    L_Last_Heartbeat_State := VI_Heartbeat_Signal;
END_IF;

// Проверка таймаута
L_Elapsed_Time := (SEL(VI_System_Time_MS >= L_Last_Heartbeat_Time, VI_System_Time_MS - L_Last_Heartbeat_Time, (4294967295 - L_Last_Heartbeat_Time) + VI_System_Time_MS + 1));

IF L_Elapsed_Time > VI_Timeout_MS THEN
    VO_Module_Online := FALSE;
    VO_Error_Active := TRUE;
ELSE
    VO_Module_Online := TRUE;
    VO_Error_Active := FALSE;
END_IF;
// >>> BULK_SYNC_ANCHOR: FB_IO_Module_Watchdog <<<
END_FUNCTION_BLOCK

(* ---- FB_Lifetime_Predictor.st ---- *)
FUNCTION_BLOCK FB_Lifetime_Predictor
VAR_INPUT
    VI_Runtime_Hours : UDINT;
    VI_Start_Count   : UDINT;
    VI_Nominal_Life  : UDINT := 10000;
END_VAR
VAR_OUTPUT
    VO_Remaining_Percent : BYTE;
    VO_Maintenance_Req   : BOOL;
END_VAR

// Упрощенная модель износа
IF VI_Nominal_Life > 0 THEN
    VO_Remaining_Percent := TO_BYTE(100 - (VI_Runtime_Hours * 100 / VI_Nominal_Life));
ELSE
    VO_Remaining_Percent := 0;
END_IF;

VO_Maintenance_Req := (VO_Remaining_Percent < 10);
END_FUNCTION_BLOCK

(* ---- FB_Lighting_Blinds_Manager.st ---- *)
FUNCTION_BLOCK FB_Lighting_Blinds_Manager
VAR_INPUT
    VI_System_Time_MS : UDINT;
    VI_IsActivePLC : BOOL;
    VI_Current_Scenario : E_SCENARIO_TYPE;
    VI_Away_Level : BYTE;
    VI_Simulation_Active : BOOL;
    VI_Is_Night : BOOL;
    VI_System_Mode : E_System_Operating_Mode;
END_VAR
VAR_IN_OUT
    VI_Manual_Light_Override : ARRAY[1..GVL_CONSTANTS.C_MAX_LIGHT_ZONES] OF BYTE;
    VI_Manual_Blinds_Override : ARRAY[1..GVL_CONSTANTS.C_MAX_BLINDS] OF BYTE;
    VI_Simulation_Lights : ARRAY[1..GVL_CONSTANTS.C_MAX_LIGHT_ZONES] OF BOOL;
    VI_Physical_Switches : ARRAY[1..GVL_CONSTANTS.C_MAX_LIGHT_ZONES] OF BOOL;
    VI_Motion_Sensors : ARRAY[1..GVL_CONSTANTS.C_MAX_LIGHT_ZONES] OF BOOL;
    VI_Rule_Actions : ARRAY[1..GVL_CONSTANTS.C_MAX_RULES] OF ST_Rule_Action;
    VI_IO_Modules_Online : ARRAY[1..GVL_CONSTANTS.C_MAX_MODULES] OF BOOL;
    VI_Wet_Zone_Map : ARRAY[1..GVL_CONSTANTS.C_MAX_LIGHT_ZONES] OF BOOL;
    VI_Scenario_Configs : ARRAY[1..GVL_CONSTANTS.C_MAX_SCENARIOS] OF ST_Scenario_Config;
END_VAR
VAR_OUTPUT
    VO_Lighting_Levels : ARRAY[1..GVL_CONSTANTS.C_MAX_LIGHT_ZONES] OF BYTE;
    VO_Blinds_Positions : ARRAY[1..GVL_CONSTANTS.C_MAX_BLINDS] OF BYTE;
    VO_Wet_Zone_Light_Active : ARRAY[1..GVL_CONSTANTS.C_MAX_WET_ZONES] OF BOOL;
END_VAR
VAR
    L_i : INT;
    L_j : INT;
    L_Base_Light : BYTE;
    L_Base_Blinds : BYTE;
    L_Target_Base_Light : BYTE;
    L_Target_Base_Blinds : BYTE;
    L_Prev_Scenario : E_SCENARIO_TYPE;
    L_Transition_Light : FB_Scenario_Transition_Controller;
    L_Transition_Blinds : FB_Scenario_Transition_Controller;
    L_Light_States : ARRAY[1..GVL_CONSTANTS.C_MAX_LIGHT_ZONES] OF BOOL;
    L_Prev_Switches : ARRAY[1..GVL_CONSTANTS.C_MAX_LIGHT_ZONES] OF BOOL;
    L_Prev_Motion_Q : ARRAY[1..GVL_CONSTANTS.C_MAX_LIGHT_ZONES] OF BOOL;
    L_Manual_Override : ARRAY[1..GVL_CONSTANTS.C_MAX_LIGHT_ZONES] OF BOOL;
    L_Motion_Timers : ARRAY[1..GVL_CONSTANTS.C_MAX_LIGHT_ZONES] OF FB_System_Timer_TOF;
    L_Rule_Light_Active : BOOL;
    L_Rule_Light_Val : BYTE;
    L_Rule_Blinds_Active : BOOL;
    L_Rule_Blinds_Val : BYTE;
    L_Wet_Zone_Idx : INT;
    L_Effective_Scenario : E_SCENARIO_TYPE;
    L_Effective_Simulation_Active : BOOL;
END_VAR

IF NOT VI_IsActivePLC THEN RETURN; END_IF;

GVL_STATE.G_Lighting_IO_Fault := FALSE;
GVL_STATE.G_Lighting_Subsystem_Degraded := FALSE;

L_Effective_Scenario := VI_Current_Scenario;
L_Effective_Simulation_Active := VI_Simulation_Active;

CASE VI_System_Mode OF
    E_System_Operating_Mode.MODE_SAFE_STOP:
        FOR L_j := 1 TO GVL_CONSTANTS.C_MAX_LIGHT_ZONES DO
            VO_Lighting_Levels[L_j] := 0;
        END_FOR;
        FOR L_j := 1 TO GVL_CONSTANTS.C_MAX_BLINDS DO
            VO_Blinds_Positions[L_j] := 100;
        END_FOR;
        FOR L_j := 1 TO GVL_CONSTANTS.C_MAX_WET_ZONES DO
            VO_Wet_Zone_Light_Active[L_j] := FALSE;
        END_FOR;
        RETURN;
    E_System_Operating_Mode.MODE_FREEZE_PROTECTION:
        L_Effective_Scenario := E_SCENARIO_TYPE.SCENARIO_NONE;
        L_Effective_Simulation_Active := FALSE;
    E_System_Operating_Mode.MODE_DEGRADED:
        L_Effective_Simulation_Active := FALSE;
END_CASE;

L_Wet_Zone_Idx := 1;
FOR L_i := 1 TO GVL_CONSTANTS.C_MAX_WET_ZONES DO
    VO_Wet_Zone_Light_Active[L_i] := FALSE;
END_FOR;

FOR L_i := 1 TO GVL_CONSTANTS.C_MAX_MODULES DO
    IF NOT VI_IO_Modules_Online[L_i] THEN
        GVL_STATE.G_Lighting_IO_Fault := TRUE;
        GVL_STATE.G_Lighting_Subsystem_Degraded := TRUE;
        FOR L_j := 1 TO GVL_CONSTANTS.C_MAX_LIGHT_ZONES DO
            VO_Lighting_Levels[L_j] := 0;
        END_FOR;
        FOR L_j := 1 TO GVL_CONSTANTS.C_MAX_BLINDS DO
            VO_Blinds_Positions[L_j] := 100;
        END_FOR;
        RETURN;
    END_IF;
END_FOR;

IF L_Effective_Scenario >= 1 AND L_Effective_Scenario <= GVL_CONSTANTS.C_MAX_SCENARIOS THEN
    L_Target_Base_Light := VI_Scenario_Configs[L_Effective_Scenario].lighting_level_base;
    L_Target_Base_Blinds := VI_Scenario_Configs[L_Effective_Scenario].blinds_position_percent;
ELSE
    L_Target_Base_Light := 100;
    L_Target_Base_Blinds := 100;
END_IF;

IF VI_Is_Night AND L_Effective_Scenario <> E_SCENARIO_TYPE.SCENARIO_AWAY AND L_Effective_Scenario <> E_SCENARIO_TYPE.SCENARIO_SLEEP THEN
    L_Target_Base_Blinds := 0;
END_IF;

IF L_Effective_Scenario <> L_Prev_Scenario THEN
    L_Transition_Light(VI_System_Time := VI_System_Time_MS, VI_Start_Time := VI_System_Time_MS, VI_Duration := 5000, VI_Start_Value := TO_REAL(L_Base_Light), VI_End_Value := TO_REAL(L_Target_Base_Light));
    L_Transition_Blinds(VI_System_Time := VI_System_Time_MS, VI_Start_Time := VI_System_Time_MS, VI_Duration := 10000, VI_Start_Value := TO_REAL(L_Base_Blinds), VI_End_Value := TO_REAL(L_Target_Base_Blinds));
    L_Prev_Scenario := L_Effective_Scenario;
ELSE
    L_Transition_Light(VI_System_Time := VI_System_Time_MS, VI_Start_Time := L_Transition_Light.VI_Start_Time, VI_Duration := L_Transition_Light.VI_Duration, VI_Start_Value := L_Transition_Light.VI_Start_Value, VI_End_Value := TO_REAL(L_Target_Base_Light));
    L_Transition_Blinds(VI_System_Time := VI_System_Time_MS, VI_Start_Time := L_Transition_Blinds.VI_Start_Time, VI_Duration := L_Transition_Blinds.VI_Duration, VI_Start_Value := L_Transition_Blinds.VI_Start_Value, VI_End_Value := TO_REAL(L_Target_Base_Blinds));
END_IF;

L_Base_Light := TO_BYTE(L_Transition_Light.VO_Current_Value);
L_Base_Blinds := TO_BYTE(L_Transition_Blinds.VO_Current_Value);

FOR L_i := 1 TO GVL_CONSTANTS.C_MAX_LIGHT_ZONES DO
    L_Rule_Light_Active := FALSE;
    L_Rule_Light_Val := 0;
    FOR L_j := 1 TO GVL_CONSTANTS.C_MAX_RULES DO
        IF VI_Rule_Actions[L_j].Active AND VI_Rule_Actions[L_j].Target_ID = L_i THEN
            IF VI_Rule_Actions[L_j].Action_Type = E_Rule_Action_Type.ACTION_SET_LIGHTING_BASE THEN
                L_Rule_Light_Active := TRUE;
                L_Rule_Light_Val := REAL_TO_BYTE(VI_Rule_Actions[L_j].Value);
                L_Light_States[L_i] := (L_Rule_Light_Val > 0);
            ELSIF VI_Rule_Actions[L_j].Action_Type = E_Rule_Action_Type.ACTION_TOGGLE_LIGHTING AND VI_Rule_Actions[L_j].Triggered THEN
                L_Light_States[L_i] := NOT L_Light_States[L_i];
            END_IF;
        END_IF;
    END_FOR;

    IF VI_Physical_Switches[L_i] AND NOT L_Prev_Switches[L_i] THEN
        L_Light_States[L_i] := NOT L_Light_States[L_i];
        L_Manual_Override[L_i] := TRUE;
    END_IF;
    L_Prev_Switches[L_i] := VI_Physical_Switches[L_i];

    L_Motion_Timers[L_i](IN := VI_Motion_Sensors[L_i], PT := T#5m, VI_System_Time_MS := VI_System_Time_MS);

    IF L_Prev_Motion_Q[L_i] AND NOT L_Motion_Timers[L_i].Q THEN
        L_Manual_Override[L_i] := FALSE;
    END_IF;
    L_Prev_Motion_Q[L_i] := L_Motion_Timers[L_i].Q;

    IF L_Motion_Timers[L_i].Q THEN
        IF NOT L_Manual_Override[L_i] THEN
            L_Light_States[L_i] := TRUE;
        END_IF;
    ELSE
        IF NOT L_Manual_Override[L_i] THEN
            L_Light_States[L_i] := FALSE;
        END_IF;
    END_IF;

    IF L_Effective_Scenario = E_SCENARIO_TYPE.SCENARIO_AWAY AND L_Effective_Simulation_Active THEN
        L_Light_States[L_i] := VI_Simulation_Lights[L_i];
    END_IF;

    IF VI_Manual_Light_Override[L_i] > 0 THEN
        VO_Lighting_Levels[L_i] := VI_Manual_Light_Override[L_i];
    ELSIF L_Rule_Light_Active THEN
        VO_Lighting_Levels[L_i] := L_Rule_Light_Val;
    ELSE
        VO_Lighting_Levels[L_i] := SEL(L_Light_States[L_i], 0, L_Base_Light);
    END_IF;

    IF VI_Wet_Zone_Map[L_i] AND L_Wet_Zone_Idx <= GVL_CONSTANTS.C_MAX_WET_ZONES THEN
        VO_Wet_Zone_Light_Active[L_Wet_Zone_Idx] := (VO_Lighting_Levels[L_i] > 10);
        L_Wet_Zone_Idx := L_Wet_Zone_Idx + 1;
    END_IF;
END_FOR;

FOR L_i := 1 TO GVL_CONSTANTS.C_MAX_BLINDS DO
    L_Rule_Blinds_Active := FALSE;
    L_Rule_Blinds_Val := 0;
    FOR L_j := 1 TO GVL_CONSTANTS.C_MAX_RULES DO
        IF VI_Rule_Actions[L_j].Active AND VI_Rule_Actions[L_j].Target_ID = L_i THEN
            IF VI_Rule_Actions[L_j].Action_Type = E_Rule_Action_Type.ACTION_SET_BLINDS THEN
                L_Rule_Blinds_Active := TRUE;
                L_Rule_Blinds_Val := REAL_TO_BYTE(VI_Rule_Actions[L_j].Value);
            END_IF;
        END_IF;
    END_FOR;

    IF VI_Manual_Blinds_Override[L_i] > 0 THEN
        VO_Blinds_Positions[L_i] := VI_Manual_Blinds_Override[L_i];
    ELSIF L_Rule_Blinds_Active THEN
        VO_Blinds_Positions[L_i] := L_Rule_Blinds_Val;
    ELSE
        VO_Blinds_Positions[L_i] := L_Base_Blinds;
    END_IF;
END_FOR;

END_FUNCTION_BLOCK
// >>> BULK_SYNC_ANCHOR: FB_Lighting_Blinds_Manager <<<

(* ---- FB_LogEvent.st ---- *)
FUNCTION_BLOCK FB_LogEvent
VAR_INPUT
    VI_Event_Type : UINT;
    VI_Timestamp  : UDINT;
    VI_Param1     : UDINT;
    VI_Param2     : UDINT;
END_VAR

GVL_EVENT.G_Event_Log[GVL_EVENT.G_Event_Head].Event_ID := GVL_EVENT.G_Event_ID_Counter;
GVL_EVENT.G_Event_Log[GVL_EVENT.G_Event_Head].Event_Type := VI_Event_Type;
GVL_EVENT.G_Event_Log[GVL_EVENT.G_Event_Head].Timestamp := VI_Timestamp;
GVL_EVENT.G_Event_Log[GVL_EVENT.G_Event_Head].Param1 := VI_Param1;
GVL_EVENT.G_Event_Log[GVL_EVENT.G_Event_Head].Param2 := VI_Param2;

GVL_EVENT.G_Event_ID_Counter := GVL_EVENT.G_Event_ID_Counter + 1;
GVL_EVENT.G_Event_Head := (GVL_EVENT.G_Event_Head + 1) MOD 64;
END_FUNCTION_BLOCK

(* ---- FB_Modbus_RTU_SysCom_Transport.st ---- *)
FUNCTION_BLOCK FB_Modbus_RTU_SysCom_Transport
VAR_INPUT
    VI_Enable : BOOL;
    VI_System_Time_MS : UDINT;
END_VAR

VAR
    L_i : INT;
END_VAR

// ======================================================
// MODBUS RTU SYSCOM TRANSPORT BOUNDARY
// ======================================================
// Byte-level transport boundary between:
//   - project RTU frame runtime
//   - concrete SysCom backend
//
// This FB intentionally does NOT:
//   - open COM ports
//   - call SysCom APIs
//   - generate fake RX frames
//   - generate fake TX done
//
// It only transfers bytes between frame runtime and SysCom backend runtime.
// ======================================================

IF NOT VI_Enable THEN

    GVL_MODBUS_SYSCOM_TRANSPORT.G_TX_Request := FALSE;
    GVL_MODBUS_SYSCOM_TRANSPORT.G_TX_Done := FALSE;
    GVL_MODBUS_SYSCOM_TRANSPORT.G_TX_Error := FALSE;
    GVL_MODBUS_SYSCOM_TRANSPORT.G_RX_Ready := FALSE;
    GVL_MODBUS_SYSCOM_TRANSPORT.G_RX_Error := FALSE;

    RETURN;
END_IF;

// ======================================================
// EXPORT TX FRAME
// ======================================================
IF GVL_MODBUS_RTU_FRAME.G_TX_Ready AND
   NOT GVL_MODBUS_SYSCOM_TRANSPORT.G_TX_Request THEN

    GVL_MODBUS_SYSCOM_TRANSPORT.G_TX_Length :=
        GVL_MODBUS_RTU_FRAME.G_TX_Frame.Length;

    FOR L_i := 0 TO 255 DO
        GVL_MODBUS_SYSCOM_TRANSPORT.G_TX_Buffer[L_i] :=
            GVL_MODBUS_RTU_FRAME.G_TX_Frame.Data[L_i];
    END_FOR;

    GVL_MODBUS_SYSCOM_TRANSPORT.G_TX_Done := FALSE;
    GVL_MODBUS_SYSCOM_TRANSPORT.G_TX_Error := FALSE;
    GVL_MODBUS_SYSCOM_TRANSPORT.G_TX_Error_Code := 0;
    GVL_MODBUS_SYSCOM_TRANSPORT.G_TX_Request := TRUE;

    GVL_MODBUS_SYSCOM_TRANSPORT.G_Last_TX_Request_MS :=
        VI_System_Time_MS;

END_IF;

// ======================================================
// CONFIRMED TX DONE - ONE SHOT CONSUME
// ======================================================
IF GVL_MODBUS_SYSCOM_TRANSPORT.G_TX_Done THEN

    GVL_MODBUS_RTU_FRAME.G_TX_Ready := FALSE;

    GVL_MODBUS_SYSCOM_TRANSPORT.G_TX_Request := FALSE;
    GVL_MODBUS_SYSCOM_TRANSPORT.G_TX_Done := FALSE;

    GVL_MODBUS_SYSCOM_TRANSPORT.G_Last_TX_Done_MS :=
        VI_System_Time_MS;

    GVL_MODBUS_SYSCOM_TRANSPORT.G_Total_TX :=
        GVL_MODBUS_SYSCOM_TRANSPORT.G_Total_TX + 1;

END_IF;

// ======================================================
// IMPORT RX FRAME - ONE SHOT CONSUME
// ======================================================
IF GVL_MODBUS_SYSCOM_TRANSPORT.G_RX_Ready THEN

    GVL_MODBUS_RTU_FRAME.G_RX_Frame.Valid := TRUE;
    GVL_MODBUS_RTU_FRAME.G_RX_Frame.Length :=
        GVL_MODBUS_SYSCOM_TRANSPORT.G_RX_Length;

    FOR L_i := 0 TO 255 DO
        GVL_MODBUS_RTU_FRAME.G_RX_Frame.Data[L_i] :=
            GVL_MODBUS_SYSCOM_TRANSPORT.G_RX_Buffer[L_i];
    END_FOR;

    GVL_MODBUS_RTU_FRAME.G_Last_RX_MS :=
        VI_System_Time_MS;

    GVL_MODBUS_RTU_FRAME.G_RX_Ready := TRUE;

    GVL_MODBUS_SYSCOM_TRANSPORT.G_Last_RX_MS :=
        VI_System_Time_MS;

    GVL_MODBUS_SYSCOM_TRANSPORT.G_Total_RX :=
        GVL_MODBUS_SYSCOM_TRANSPORT.G_Total_RX + 1;

    GVL_MODBUS_SYSCOM_TRANSPORT.G_RX_Ready := FALSE;

END_IF;

// ======================================================
// TRANSPORT ERRORS - ONE SHOT CONSUME
// ======================================================
IF GVL_MODBUS_SYSCOM_TRANSPORT.G_TX_Error OR
   GVL_MODBUS_SYSCOM_TRANSPORT.G_RX_Error THEN

    GVL_MODBUS_SYSCOM_TRANSPORT.G_Total_Errors :=
        GVL_MODBUS_SYSCOM_TRANSPORT.G_Total_Errors + 1;

    GVL_MODBUS_SYSCOM_TRANSPORT.G_TX_Error := FALSE;
    GVL_MODBUS_SYSCOM_TRANSPORT.G_RX_Error := FALSE;

END_IF;

END_FUNCTION_BLOCK

(* ---- FB_Presence_Playback.st ---- *)
FUNCTION_BLOCK FB_Presence_Playback
VAR_INPUT
    VI_Mode_Record : BOOL;
    VI_Time_Index   : UDINT;
END_VAR
VAR_IN_OUT
    VI_Light_Inputs : ARRAY[1..32] OF BOOL;
END_VAR
VAR_OUTPUT
    VO_Light_Outputs : ARRAY[1..32] OF BOOL;
END_VAR
VAR
    L_Current_Slot : UDINT;
    L_i : INT;
END_VAR

L_Current_Slot := (VI_Time_Index / (GVL_CONSTANTS.C_MS_IN_MINUTE * 10)) MOD TO_UDINT(GVL_CONSTANTS.C_MAX_PRESENCE_HISTORY);

IF VI_Mode_Record THEN
    GVL_Retain.G_Presence_History[L_Current_Slot] := 0;
    FOR L_i := 1 TO 32 DO
        IF VI_Light_Inputs[L_i] THEN
            GVL_Retain.G_Presence_History[L_Current_Slot] := GVL_Retain.G_Presence_History[L_Current_Slot] OR SHL(WORD#1, L_i-1);
        END_IF;
    END_FOR;
ELSE
    FOR L_i := 1 TO 32 DO
        VO_Light_Outputs[L_i] := (GVL_Retain.G_Presence_History[L_Current_Slot] AND SHL(WORD#1, L_i-1)) <> 0;
    END_FOR;
END_IF;

END_FUNCTION_BLOCK

(* ---- FB_Runtime_Restart_Continuity.st ---- *)
FUNCTION_BLOCK FB_Runtime_Restart_Continuity
VAR_INPUT
    VI_Enable : BOOL;
    VI_System_Time_MS : UDINT;
    VI_Warm_Restart : BOOL;
END_VAR
VAR
    L_State : ST_Runtime_Restart_Continuity_State;
END_VAR

IF NOT VI_Enable THEN
    GVL_Runtime_Restart_Continuity.G_Runtime_Valid := FALSE;
    RETURN;
END_IF;

L_State.Runtime_Valid := TRUE;
L_State.Runtime_System_Time_MS := VI_System_Time_MS;

L_State.Warm_Restart_Detected := VI_Warm_Restart;
L_State.Cold_Start_Detected := NOT VI_Warm_Restart;

L_State.Active_Config_Version :=
    GVL_Water_Topology_Config.G_Active_Config_Version;

L_State.Restored_Config_Version :=
    GVL_Runtime_Restart_Continuity.G_Last_Stable_Config_Version;

L_State.Last_Stable_Config_Version :=
    GVL_Runtime_Restart_Continuity.G_Last_Stable_Config_Version;

L_State.Restore_Requested :=
    GVL_Runtime_Restart_Continuity.G_Restore_Request;

L_State.Post_Restart_Validation_Required :=
    GVL_Runtime_Restart_Continuity.G_Post_Restart_Validation_Request;

L_State.Retained_State_Valid := TRUE;
L_State.Topology_Restore_Valid := TRUE;
L_State.Config_Restore_Valid := TRUE;
L_State.Recovery_Restore_Valid := TRUE;
L_State.Quarantine_Restore_Valid := TRUE;

IF L_State.Restore_Requested THEN

    IF L_State.Retained_State_Valid
       AND L_State.Topology_Restore_Valid
       AND L_State.Config_Restore_Valid THEN

        L_State.Restore_Allowed := TRUE;
        L_State.Restore_Completed := TRUE;

        GVL_Config_Activation.G_Config_Quarantine_Active :=
            GVL_Runtime_Restart_Continuity.G_Last_Known_Quarantine_State;

        L_State.Status_Code := 1;
        L_State.Status_Text := 'Runtime continuity restored';

    ELSE

        L_State.Restore_Blocked := TRUE;
        L_State.Safe_Mode_Required := TRUE;
        L_State.Operator_Ack_Required := TRUE;

        L_State.Status_Code := 2;
        L_State.Status_Text := 'Runtime continuity restore blocked';

    END_IF;

ELSIF L_State.Post_Restart_Validation_Required THEN

    IF GVL_Water_Runtime_Hardening.G_Runtime_Valid
       AND GVL_Water_Output_Reconciliation.G_Runtime_Valid
       AND NOT GVL_Water_Output_Reconciliation.G_Any_Conflict_Detected THEN

        L_State.Post_Restart_Validation_OK := TRUE;

        L_State.Status_Code := 0;
        L_State.Status_Text := 'Post-restart validation healthy';

    ELSE

        L_State.Post_Restart_Validation_Failed := TRUE;
        L_State.Safe_Mode_Required := TRUE;

        L_State.Status_Code := 3;
        L_State.Status_Text := 'Post-restart validation failed';

    END_IF;

ELSE

    L_State.Status_Code := 0;
    L_State.Status_Text := 'Runtime restart continuity healthy';

END_IF;

GVL_Runtime_Restart_Continuity.G_Continuity_State := L_State;

GVL_Runtime_Restart_Continuity.G_Runtime_Valid := TRUE;
GVL_Runtime_Restart_Continuity.G_Last_Update_MS := VI_System_Time_MS;
GVL_Runtime_Restart_Continuity.G_Status_Code := L_State.Status_Code;
GVL_Runtime_Restart_Continuity.G_Status_Text := L_State.Status_Text;

END_FUNCTION_BLOCK

(* ---- FB_SHA1.st ---- *)
FUNCTION_BLOCK FB_SHA1
VAR_INPUT
    Length : INT;
END_VAR
VAR_IN_OUT
    Data : ARRAY[0..127] OF BYTE;
END_VAR
VAR_OUTPUT
    Hash : ARRAY[0..19] OF BYTE;
END_VAR
VAR
    H0, H1, H2, H3, H4 : DWORD;
    A, B, C, D, E, F, K, Temp : DWORD;
    W : ARRAY[0..79] OF DWORD;
    i, j, t : INT;
    PaddedData : ARRAY[0..127] OF BYTE;
    PaddedLength : INT;
    NumBlocks : INT;
    BlockOffset : INT;
END_VAR

// Initialize variables
H0 := 16#67452301;
H1 := 16#EFCDAB89;
H2 := 16#98BADCFE;
H3 := 16#10325476;
H4 := 16#C3D2E1F0;

// Pre-processing
FOR i := 0 TO Length - 1 DO
    PaddedData[i] := Data[i];
END_FOR;

// Append the bit '1' to the message
PaddedData[Length] := 16#80;

// Append 0 <= k < 512 bits '0', such that the resulting message length in bits
// is congruent to -64 ≡ 448 (mod 512)
PaddedLength := Length + 1;
WHILE (PaddedLength MOD 64) <> 56 DO
    PaddedData[PaddedLength] := 0;
    PaddedLength := PaddedLength + 1;
END_WHILE;

// Append length of message (before pre-processing), in bits, as 64-bit big-endian integer
// Since our message is small (max 127 bytes), we only need the lower 32 bits
Temp := TO_DWORD(Length * 8);
PaddedData[PaddedLength] := 0;
PaddedData[PaddedLength+1] := 0;
PaddedData[PaddedLength+2] := 0;
PaddedData[PaddedLength+3] := 0;
PaddedData[PaddedLength+4] := TO_BYTE(SHR(Temp, 24));
PaddedData[PaddedLength+5] := TO_BYTE(SHR(Temp, 16));
PaddedData[PaddedLength+6] := TO_BYTE(SHR(Temp, 8));
PaddedData[PaddedLength+7] := TO_BYTE(Temp);
PaddedLength := PaddedLength + 8;

NumBlocks := PaddedLength / 64;

// Process the message in successive 512-bit chunks
FOR i := 0 TO NumBlocks - 1 DO
    BlockOffset := i * 64;

    // Break chunk into sixteen 32-bit big-endian words w[i], 0 <= i <= 15
    FOR j := 0 TO 15 DO
        W[j] := SHL(TO_DWORD(PaddedData[BlockOffset + j*4]), 24) OR
                SHL(TO_DWORD(PaddedData[BlockOffset + j*4 + 1]), 16) OR
                SHL(TO_DWORD(PaddedData[BlockOffset + j*4 + 2]), 8) OR
                TO_DWORD(PaddedData[BlockOffset + j*4 + 3]);
    END_FOR;

    // Message schedule: extend the sixteen 32-bit words into eighty 32-bit words
    FOR j := 16 TO 79 DO
        Temp := W[j-3] XOR W[j-8] XOR W[j-14] XOR W[j-16];
        W[j] := SHL(Temp, 1) OR SHR(Temp, 31); // Left rotate by 1
    END_FOR;

    // Initialize hash value for this chunk
    A := H0;
    B := H1;
    C := H2;
    D := H3;
    E := H4;

    // Main loop
    FOR j := 0 TO 79 DO
        IF j <= 19 THEN
            F := (B AND C) OR ((NOT B) AND D);
            K := 16#5A827999;
        ELSIF j <= 39 THEN
            F := B XOR C XOR D;
            K := 16#6ED9EBA1;
        ELSIF j <= 59 THEN
            F := (B AND C) OR (B AND D) OR (C AND D);
            K := 16#8F1BBCDC;
        ELSE
            F := B XOR C XOR D;
            K := 16#CA62C1D6;
        END_IF;

        Temp := (SHL(A, 5) OR SHR(A, 27)) + F + E + K + W[j];
        E := D;
        D := C;
        C := SHL(B, 30) OR SHR(B, 2);
        B := A;
        A := Temp;
    END_FOR;

    // Add this chunk's hash to result so far
    H0 := H0 + A;
    H1 := H1 + B;
    H2 := H2 + C;
    H3 := H3 + D;
    H4 := H4 + E;
END_FOR;

// Produce the final hash value (big-endian)
Hash[0] := TO_BYTE(SHR(H0, 24)); Hash[1] := TO_BYTE(SHR(H0, 16)); Hash[2] := TO_BYTE(SHR(H0, 8)); Hash[3] := TO_BYTE(H0);
Hash[4] := TO_BYTE(SHR(H1, 24)); Hash[5] := TO_BYTE(SHR(H1, 16)); Hash[6] := TO_BYTE(SHR(H1, 8)); Hash[7] := TO_BYTE(H1);
Hash[8] := TO_BYTE(SHR(H2, 24)); Hash[9] := TO_BYTE(SHR(H2, 16)); Hash[10] := TO_BYTE(SHR(H2, 8)); Hash[11] := TO_BYTE(H2);
Hash[12] := TO_BYTE(SHR(H3, 24)); Hash[13] := TO_BYTE(SHR(H3, 16)); Hash[14] := TO_BYTE(SHR(H3, 8)); Hash[15] := TO_BYTE(H3);
Hash[16] := TO_BYTE(SHR(H4, 24)); Hash[17] := TO_BYTE(SHR(H4, 16)); Hash[18] := TO_BYTE(SHR(H4, 8)); Hash[19] := TO_BYTE(H4);
END_FUNCTION_BLOCK

(* ---- FB_Socket_Manager.st ---- *)
FUNCTION_BLOCK FB_Socket_Manager
// Менеджер управления розетками.
// Обеспечивает работу по сценариям, правилам и аварийное отключение (без локальных выключателей розеток).
VAR_INPUT
    VI_System_Time_MS : UDINT; // Системное время в миллисекундах
    VI_IsActivePLC : BOOL; // Флаг активности ПЛК (TRUE = ведущий)
    VI_Scenario : E_SCENARIO_TYPE; // Текущий глобальный сценарий
    VI_Fire_Alarm : BOOL; // Флаг пожарной тревоги
    VI_Flood_Alarm : BOOL; // Флаг тревоги протечки
    VI_Security_Armed : BOOL; // Состояние охраны (TRUE = включена)
END_VAR
VAR_IN_OUT
    VI_Manual_Override : ARRAY[1..GVL_CONSTANTS.C_MAX_SOCKETS] OF BOOL; // Ручное переопределение состояния (HMI)
    VI_Physical_Switches : ARRAY[1..GVL_CONSTANTS.C_MAX_SOCKETS] OF BOOL; // Legacy-вход: не используется в текущей концепции
    VI_Rule_Actions : ARRAY[1..GVL_CONSTANTS.C_MAX_RULES] OF ST_Rule_Action; // Действия от Rule Engine
    VI_IO_Modules_Online : ARRAY[1..GVL_CONSTANTS.C_MAX_MODULES] OF BOOL; // Статусы модулей ввода-вывода
END_VAR
VAR_OUTPUT
    VO_Socket_States : ARRAY[1..GVL_CONSTANTS.C_MAX_SOCKETS] OF BOOL; // Выходные состояния розеток
    VO_Internal_States : ARRAY[1..GVL_CONSTANTS.C_MAX_SOCKETS] OF BOOL; // Внутренние состояния для репликации
END_VAR
VAR
    L_i : INT;
    L_j : INT;
    L_Rule_State : BOOL;
    L_Rule_Active : BOOL;
    L_Internal_State : ARRAY[1..GVL_CONSTANTS.C_MAX_SOCKETS] OF BOOL;
    L_Manual_Trig : ARRAY[1..GVL_CONSTANTS.C_MAX_SOCKETS] OF R_TRIG;
END_VAR

IF NOT VI_IsActivePLC THEN RETURN; END_IF;

// Проверка связи с модулями ввода-вывода
FOR L_i := 1 TO GVL_CONSTANTS.C_MAX_MODULES DO
    IF NOT VI_IO_Modules_Online[L_i] THEN
        // Переход в безопасное состояние при потере связи (отключение всех розеток)
        FOR L_j := 1 TO GVL_CONSTANTS.C_MAX_SOCKETS DO
            VO_Socket_States[L_j] := FALSE;
        END_FOR;
        RETURN;
    END_IF;
END_FOR;

FOR L_i := 1 TO GVL_CONSTANTS.C_MAX_SOCKETS DO
    L_Rule_Active := FALSE;
    L_Rule_State := FALSE;

    L_Manual_Trig[L_i](CLK := VI_Manual_Override[L_i]);

    // Ручное переключение
    IF L_Manual_Trig[L_i].Q THEN
        L_Internal_State[L_i] := NOT L_Internal_State[L_i];
    END_IF;

    // Проверка правил для текущей розетки
    FOR L_j := 1 TO GVL_CONSTANTS.C_MAX_RULES DO
        IF VI_Rule_Actions[L_j].Active AND VI_Rule_Actions[L_j].Target_ID = L_i THEN
            IF VI_Rule_Actions[L_j].Action_Type = E_Rule_Action_Type.ACTION_SET_SOCKET THEN
                L_Rule_Active := TRUE;
                L_Rule_State := (VI_Rule_Actions[L_j].Value > 0.5);
                L_Internal_State[L_i] := L_Rule_State; // Синхронизация внутреннего состояния
            ELSIF VI_Rule_Actions[L_j].Action_Type = E_Rule_Action_Type.ACTION_TOGGLE_SOCKET AND VI_Rule_Actions[L_j].Triggered THEN
                L_Internal_State[L_i] := NOT L_Internal_State[L_i]; // Toggle
            END_IF;
        END_IF;
    END_FOR;

    // Аварийное отключение
    IF VI_Fire_Alarm OR VI_Flood_Alarm THEN
        // Розетки 1-4 неотключаемые (холодильник, сервер и т.д.)
        IF L_i > 4 THEN
            VO_Socket_States[L_i] := FALSE;
        ELSE
            // Критические розетки сохраняют свое текущее внутреннее состояние, а не форсируются в TRUE
            VO_Socket_States[L_i] := L_Internal_State[L_i];
        END_IF;
    ELSIF VI_Scenario = E_SCENARIO_TYPE.SCENARIO_AWAY OR VI_Security_Armed THEN
        // Master Off
        IF L_i > 4 THEN
            VO_Socket_States[L_i] := FALSE;
        ELSE
            // Неотключаемые розетки могут управляться вручную
            VO_Socket_States[L_i] := L_Internal_State[L_i];
        END_IF;
    ELSE
        // Нормальный режим: состояние определяется внутренним состоянием (ручным или правилом)
        IF L_Rule_Active THEN
            VO_Socket_States[L_i] := L_Rule_State;
        ELSE
            VO_Socket_States[L_i] := L_Internal_State[L_i];
        END_IF;
    END_IF;
END_FOR;

VO_Internal_States := L_Internal_State;

END_FUNCTION_BLOCK
// >>> BULK_SYNC_ANCHOR: FB_Socket_Manager <<<

(* ---- FB_System_Diagnostics_Publisher.st ---- *)
FUNCTION_BLOCK FB_System_Diagnostics_Publisher
VAR_INPUT
    VI_Enable : BOOL;
    VI_System_Time_MS : UDINT;
    VI_Backup_Pump_Out_Of_Service : BOOL;
    VI_Electric_Heater_Out_Of_Service : BOOL;
    VI_Manifold_Pump_Out_Of_Service : ARRAY[1..GVL_CONSTANTS.C_MAX_MANIFOLDS] OF BOOL;
    VI_DHW_Heating_Pump_Out_Of_Service : BOOL;
    VI_DHW_Circ_Pump_Out_Of_Service : BOOL;
    VI_User_Access_Level : INT;
    VI_Dangerous_Action_Pending : BOOL;
    VI_Dangerous_Action_Text : STRING(160);
    VI_Sensor_Fault : BOOL;
    VI_IO_Offline : BOOL;
    VI_Subsystem_Degraded : BOOL;
    VI_Manifold_Pressure_Fault : ARRAY[1..GVL_CONSTANTS.C_MAX_MANIFOLDS] OF BOOL;
    VI_Manifold_Current_Fault : ARRAY[1..GVL_CONSTANTS.C_MAX_MANIFOLDS] OF BOOL;
    VI_Manifold_Return_Temp_Fault : ARRAY[1..GVL_CONSTANTS.C_MAX_MANIFOLDS] OF BOOL;
END_VAR
VAR_OUTPUT
    VO_Diagnostics : ST_System_Diagnostics;
    VO_Publication_Valid : BOOL;
    VO_Status_Code : UINT;
    VO_Status_Text : STRING(128);
END_VAR
VAR
    L_i : INT;
    L_Pressure_First : INT;
    L_Current_First : INT;
    L_Return_First : INT;
    L_Any_Manifold_Fault : BOOL;
END_VAR

VO_Diagnostics.Freeze_Hardware_Event_Pending := FALSE;
VO_Diagnostics.Freeze_Hardware_Event_Text := '';
VO_Diagnostics.Backup_Pump_Fault := VI_Backup_Pump_Out_Of_Service;
VO_Diagnostics.Electric_Heater_Fault := VI_Electric_Heater_Out_Of_Service;
VO_Diagnostics.Backup_Pump_Recovered_After_Retry := FALSE;
VO_Diagnostics.Electric_Heater_Recovered_After_Retry := FALSE;
VO_Diagnostics.Backup_Pump_Out_Of_Service := VI_Backup_Pump_Out_Of_Service;
VO_Diagnostics.Electric_Heater_Out_Of_Service := VI_Electric_Heater_Out_Of_Service;

VO_Diagnostics.Pump_Exercise_Active := FALSE;
VO_Diagnostics.Pump_Exercise_Failed := FALSE;
VO_Diagnostics.Pump_Exercise_Last_Equipment := '';
VO_Diagnostics.Pump_Exercise_Last_Result := 'Pump exercise publisher passive';
VO_Diagnostics.Pump_Exercise_No_Feedback_Count := 0;
VO_Diagnostics.DHW_Heating_Pump_Exercise_Count := 0;
VO_Diagnostics.DHW_Circ_Pump_Exercise_Count := 0;
VO_Diagnostics.Backup_Pump_Exercise_Count := 0;
VO_Diagnostics.Pump_Exercise_Event_Seq := VI_System_Time_MS;
VO_Diagnostics.Pump_Exercise_Journal_1 := 'Passive diagnostics publication active';
VO_Diagnostics.Pump_Exercise_Journal_2 := '';
VO_Diagnostics.Pump_Exercise_Journal_3 := '';
VO_Diagnostics.Pump_Exercise_Journal_Last_Seq := VI_System_Time_MS;

VO_Diagnostics.Pump_Maintenance_Required := VI_Backup_Pump_Out_Of_Service OR VI_Electric_Heater_Out_Of_Service;
VO_Diagnostics.Pump_Maintenance_Warning := VO_Diagnostics.Pump_Maintenance_Required;

VO_Diagnostics.DHW_Heating_Pump_Out_Of_Service := VI_DHW_Heating_Pump_Out_Of_Service;
VO_Diagnostics.DHW_Circ_Pump_Out_Of_Service := VI_DHW_Circ_Pump_Out_Of_Service;

VO_Diagnostics.Maintenance_Last_Action := 'Diagnostics publication only';
VO_Diagnostics.Operator_Action_Blocked := FALSE;
VO_Diagnostics.Operator_Block_Reason := '';
VO_Diagnostics.Operator_Last_Forbidden_Action := '';
VO_Diagnostics.Operator_Journal_1 := 'Operator diagnostics passive';
VO_Diagnostics.Operator_Journal_2 := '';
VO_Diagnostics.Operator_Journal_3 := '';
VO_Diagnostics.Operator_Journal_Event_Seq := VI_System_Time_MS;
VO_Diagnostics.Operator_Journal_Last_Seq := VI_System_Time_MS;

VO_Diagnostics.Dangerous_Action_Pending_Confirm := VI_Dangerous_Action_Pending;
VO_Diagnostics.Dangerous_Action_Confirm_Text := VI_Dangerous_Action_Text;
VO_Diagnostics.Dangerous_Action_Confirm_Deadline_MS := 0;
VO_Diagnostics.User_Access_Level_Active := VI_User_Access_Level;
VO_Diagnostics.User_Access_Denied := FALSE;
VO_Diagnostics.User_Access_Deny_Reason := '';

VO_Diagnostics.Valve_Test_Mode_Active := FALSE;
VO_Diagnostics.Valve_Test_Deadline_MS := 0;
VO_Diagnostics.Valve_Test_Remaining_MS := 0;
VO_Diagnostics.Valve_Test_Validation_OK := TRUE;
VO_Diagnostics.Valve_Test_Validation_Text := 'No generic valve test active';
VO_Diagnostics.Valve_Test_Forced_Close := FALSE;

VO_Diagnostics.Water_Valve_Test_Mode_Active := FALSE;
VO_Diagnostics.Water_Valve_Test_Deadline_MS := 0;
VO_Diagnostics.Water_Valve_Test_Remaining_MS := 0;
VO_Diagnostics.Water_Valve_Test_Validation_OK := TRUE;
VO_Diagnostics.Water_Valve_Test_Validation_Text := 'No water valve test active';
VO_Diagnostics.Water_Valve_Test_Forced_Close := FALSE;
VO_Diagnostics.Gas_Valve_Test_Mode_Active := FALSE;
VO_Diagnostics.Gas_Valve_Test_Deadline_MS := 0;
VO_Diagnostics.Gas_Valve_Test_Remaining_MS := 0;
VO_Diagnostics.Gas_Valve_Test_Validation_OK := TRUE;
VO_Diagnostics.Gas_Valve_Test_Validation_Text := 'No gas valve test active';
VO_Diagnostics.Gas_Valve_Test_Forced_Close := FALSE;

VO_Diagnostics.Active_Leak_Sensor_Index := 0;
VO_Diagnostics.Active_Gas_Sensor_Index := 0;
VO_Diagnostics.Active_Leak_Zone_Name := '';
VO_Diagnostics.Active_Gas_Zone_Name := '';
VO_Diagnostics.Water_Valve_Test_Context := 'Water diagnostics passive';
VO_Diagnostics.Gas_Valve_Test_Context := 'Gas diagnostics passive';

VO_Diagnostics.Water_Recovery_Target_Zone_Index := 0;
VO_Diagnostics.Gas_Recovery_Target_Zone_Index := 0;
VO_Diagnostics.Water_Recovery_Selective_Allowed := FALSE;
VO_Diagnostics.Gas_Recovery_Selective_Allowed := FALSE;
VO_Diagnostics.Water_Recovery_Selective_Text := 'Selective water recovery inactive';
VO_Diagnostics.Gas_Recovery_Selective_Text := 'Selective gas recovery inactive';
VO_Diagnostics.Water_Recovery_Physical_Active := FALSE;
VO_Diagnostics.Water_Recovery_Physical_Zone_Name := '';

VO_Diagnostics.Water_Valve_Exercise_Last_Zone := 0;
VO_Diagnostics.Water_Valve_Exercise_Last_Result := 'Water valve exercise inactive';
VO_Diagnostics.Water_Close_Fault_Active := FALSE;
VO_Diagnostics.Water_Close_Fault_Zone_Name := '';
VO_Diagnostics.Water_Close_Fault_Text := '';
VO_Diagnostics.Water_Localization_Failed := FALSE;
VO_Diagnostics.Water_Main_Shutdown_Recommended := FALSE;
VO_Diagnostics.Water_Escalation_Text := '';
VO_Diagnostics.Alarm_Event_Pulse := FALSE;
VO_Diagnostics.Alarm_Event_Code := 0;
VO_Diagnostics.Alarm_Event_Value := 0.0;
VO_Diagnostics.Sensor_Fault := VI_Sensor_Fault;
VO_Diagnostics.IO_Offline := VI_IO_Offline;
VO_Diagnostics.Subsystem_Degraded := VI_Subsystem_Degraded;

L_Pressure_First := 0;
L_Current_First := 0;
L_Return_First := 0;
L_Any_Manifold_Fault := FALSE;

FOR L_i := 1 TO GVL_CONSTANTS.C_MAX_MANIFOLDS DO
    VO_Diagnostics.Manifold_Pump_Out_Of_Service[L_i] := VI_Manifold_Pump_Out_Of_Service[L_i];
    VO_Diagnostics.Manifold_Pump_Exercise_Count[L_i] := 0;

    VO_Diagnostics.Manifold_Pressure_Fault[L_i] := VI_Manifold_Pressure_Fault[L_i];
    VO_Diagnostics.Manifold_Pressure_Diag_Code[L_i] := SEL(VI_Manifold_Pressure_Fault[L_i], WORD#0, WORD#16#E004);
    IF VI_Manifold_Pressure_Fault[L_i] AND (L_Pressure_First = 0) THEN
        L_Pressure_First := L_i;
    END_IF;

    VO_Diagnostics.Manifold_Current_Fault[L_i] := VI_Manifold_Current_Fault[L_i];
    VO_Diagnostics.Manifold_Current_Diag_Code[L_i] := SEL(VI_Manifold_Current_Fault[L_i], WORD#0, WORD#16#E00A);
    IF VI_Manifold_Current_Fault[L_i] AND (L_Current_First = 0) THEN
        L_Current_First := L_i;
    END_IF;

    VO_Diagnostics.Manifold_Return_Temp_Fault[L_i] := VI_Manifold_Return_Temp_Fault[L_i];
    VO_Diagnostics.Manifold_Return_Temp_Diag_Code[L_i] := SEL(VI_Manifold_Return_Temp_Fault[L_i], WORD#0, WORD#16#E00D);
    IF VI_Manifold_Return_Temp_Fault[L_i] AND (L_Return_First = 0) THEN
        L_Return_First := L_i;
    END_IF;

    VO_Diagnostics.Manifold_Sensor_Fault_Count[L_i] := 0;
    IF VI_Manifold_Pressure_Fault[L_i] THEN
        VO_Diagnostics.Manifold_Sensor_Fault_Count[L_i] := VO_Diagnostics.Manifold_Sensor_Fault_Count[L_i] + 1;
    END_IF;
    IF VI_Manifold_Current_Fault[L_i] THEN
        VO_Diagnostics.Manifold_Sensor_Fault_Count[L_i] := VO_Diagnostics.Manifold_Sensor_Fault_Count[L_i] + 1;
    END_IF;
    IF VI_Manifold_Return_Temp_Fault[L_i] THEN
        VO_Diagnostics.Manifold_Sensor_Fault_Count[L_i] := VO_Diagnostics.Manifold_Sensor_Fault_Count[L_i] + 1;
    END_IF;

    VO_Diagnostics.Manifold_Sensor_Out_Of_Service[L_i] := VO_Diagnostics.Manifold_Sensor_Fault_Count[L_i] > 0;
    L_Any_Manifold_Fault := L_Any_Manifold_Fault OR VO_Diagnostics.Manifold_Sensor_Out_Of_Service[L_i];
END_FOR;

FOR L_i := 1 TO 32 DO
    VO_Diagnostics.Water_Zone_Open_Fault[L_i] := FALSE;
    VO_Diagnostics.Water_Zone_Close_Fault[L_i] := FALSE;
    VO_Diagnostics.Water_Zone_Critical_Close_Fault[L_i] := FALSE;
    VO_Diagnostics.Water_Zone_Close_Retry_Active[L_i] := FALSE;
    VO_Diagnostics.Water_Zone_Close_Retry_Count[L_i] := 0;
    VO_Diagnostics.Water_Zone_Close_Recovered_After_Retry[L_i] := FALSE;
END_FOR;

VO_Diagnostics.Manifold_Pressure_Fault_Active := L_Pressure_First > 0;
VO_Diagnostics.Manifold_Pressure_First_Fault_Index := L_Pressure_First;
VO_Diagnostics.Manifold_Pressure_Fault_Text := SEL(L_Pressure_First > 0, '', 'Manifold pressure fault active');

VO_Diagnostics.Manifold_Current_Fault_Active := L_Current_First > 0;
VO_Diagnostics.Manifold_Current_First_Fault_Index := L_Current_First;
VO_Diagnostics.Manifold_Current_Fault_Text := SEL(L_Current_First > 0, '', 'Manifold current fault active');

VO_Diagnostics.Manifold_Return_Temp_Fault_Active := L_Return_First > 0;
VO_Diagnostics.Manifold_Return_Temp_First_Fault_Index := L_Return_First;
VO_Diagnostics.Manifold_Return_Temp_Fault_Text := SEL(L_Return_First > 0, '', 'Manifold return temperature fault active');

VO_Diagnostics.Manifold_Sensor_Out_Of_Service_Active := L_Any_Manifold_Fault;
VO_Diagnostics.Manifold_Sensor_First_OOS_Index := SEL(L_Pressure_First > 0, SEL(L_Current_First > 0, L_Return_First, L_Current_First), L_Pressure_First);
VO_Diagnostics.Manifold_Sensor_OOS_Text := SEL(L_Any_Manifold_Fault, '', 'Manifold sensor out of service');

VO_Publication_Valid := VI_Enable;
VO_Status_Code := SEL(VI_Subsystem_Degraded OR VI_IO_Offline OR VI_Sensor_Fault OR L_Any_Manifold_Fault, 1, 900);
VO_Status_Text := SEL(VO_Status_Code = 1, 'System diagnostics nominal', 'System diagnostics degraded');

END_FUNCTION_BLOCK
// >>> BULK_SYNC_ANCHOR: FB_System_Diagnostics_Publisher <<<

(* ---- FB_System_Evacuation.st ---- *)
// ==============================================================================
// System evacuation helper
//
// Internal helper for PRG_System.
// Owns evacuation guidance, target/hazard zone name projection,
// and evacuation lighting activation.
// ==============================================================================
FUNCTION_BLOCK FB_System_Evacuation
VAR
    L_i : INT;
END_VAR

FOR L_i := 1 TO 32 DO
    GVL_STATE.G_Evac_Guidance[L_i] := 0;

    IF GVL_STATE.G_Evac_Hazard_Zone[L_i] THEN
        GVL_STATE.G_Evac_Guidance[L_i] := -1;
    END_IF;

    IF GVL_CONFIG.G_Evac_Exit_Zones[L_i] AND NOT GVL_STATE.G_Evac_Hazard_Zone[L_i] THEN
        GVL_STATE.G_Evac_Guidance[L_i] := 1;
    END_IF;
END_FOR;

GVL_STATUS.G_Evac_Target_Zone_Name := '';
GVL_STATUS.G_Evac_Hazard_Zone_Name := '';

FOR L_i := 1 TO 32 DO
    IF (GVL_STATUS.G_Evac_Hazard_Zone_Name = '') AND GVL_STATE.G_Evac_Hazard_Zone[L_i] THEN
        GVL_STATUS.G_Evac_Hazard_Zone_Name := GVL_CONFIG.G_Evac_Zone_Names[L_i];
        IF GVL_STATUS.G_Evac_Hazard_Zone_Name = '' THEN
            GVL_STATUS.G_Evac_Hazard_Zone_Name := CONCAT('Zone ', INT_TO_STRING(L_i));
        END_IF;
    END_IF;

    IF (GVL_STATUS.G_Evac_Target_Zone_Name = '') AND (GVL_STATE.G_Evac_Guidance[L_i] = 1) THEN
        GVL_STATUS.G_Evac_Target_Zone_Name := GVL_CONFIG.G_Evac_Zone_Names[L_i];
        IF GVL_STATUS.G_Evac_Target_Zone_Name = '' THEN
            GVL_STATUS.G_Evac_Target_Zone_Name := CONCAT('Zone ', INT_TO_STRING(L_i));
        END_IF;
    END_IF;
END_FOR;

IF GVL_STATE.G_System_Mode = E_System_Operating_Mode.MODE_SAFE_STOP AND GVL_STATE.G_Safety_Smoke_Latched THEN
    GVL_STATE.G_Evacuation_Lighting_Active := TRUE;
ELSE
    GVL_STATE.G_Evacuation_Lighting_Active := FALSE;
END_IF;

// >>> BULK_SYNC_ANCHOR: FB_System_Evacuation <<<
END_FUNCTION_BLOCK

(* ---- FB_System_Gateway_Intent.st ---- *)
FUNCTION_BLOCK FB_System_Gateway_Intent
VAR_INPUT
    VI_System_Time_MS : UDINT;
    VI_IsActivePLC : BOOL;
    VI_Gateway_Writes_Allowed : BOOL;
END_VAR

VAR_IN_OUT
    VIO_FloorHeating_Temps : ARRAY[1..GVL_CONSTANTS.C_MAX_HEATING_CIRCUITS] OF REAL;
    VIO_Zone_Valve_States : ARRAY[1..GVL_CONSTANTS.C_MAX_HEATING_CIRCUITS] OF BOOL;
    VIO_Lighting_Base_Levels : ARRAY[1..GVL_CONSTANTS.C_MAX_LIGHT_ZONES] OF BYTE;
    VIO_Scenario_Req_Gateway : E_SCENARIO_TYPE;
END_VAR

VAR
    fbGateway : FB_Gateway_Interface;
    L_Gateway_Flood_Alarm_Active : BOOL;
    L_Gateway_Gas_Alarm_Active : BOOL;
    L_Gateway_Fire_Alarm_Active : BOOL;
END_VAR

// Gateway telemetry must expose authoritative safety truth and latches,
// not stale alarm projection fields.
L_Gateway_Flood_Alarm_Active := GVL_HEALTH_BRIDGE.G_Leak_Detected OR GVL_STATE.G_Safety_Leak_Latched;
L_Gateway_Gas_Alarm_Active := GVL_HEALTH_BRIDGE.G_Gas_Detected OR GVL_HEALTH_BRIDGE.G_CO_Alarm_Level OR GVL_STATE.G_Safety_Gas_Latched;
L_Gateway_Fire_Alarm_Active := GVL_HEALTH_BRIDGE.G_Smoke_Detected OR GVL_STATE.G_Safety_Smoke_Latched;

fbGateway(
    VI_System_Time_MS := VI_System_Time_MS,
    VI_Local_PLC_Role := SEL(VI_IsActivePLC, E_PLC_ROLE.ROLE_STANDBY, E_PLC_ROLE.ROLE_ACTIVE),
    VI_Incoming_Command := GVL_GATEWAY.G_Gateway_Command,
    VI_Command_Received := GVL_GATEWAY.G_Gateway_Command_Received,
    VI_FloorHeating_Temps := VIO_FloorHeating_Temps,
    VI_Room_Temps := GVL_STATE.G_Room_Temps,
    VI_Zone_Valve_States := VIO_Zone_Valve_States,
    VI_Manifold_Pressures := GVL_STATE.G_Manifold_Pressures,
    VI_Manifold_Pump_States := GVL_STATE.G_Manifold_Pumps,
    VI_Outdoor_Temp := GVL_STATE.G_Outdoor_Temp,
    VI_Security_Armed := GVL_ALARM.G_Security_Armed,
    VI_Flood_Alarm_Active := L_Gateway_Flood_Alarm_Active,
    VI_Gas_Alarm_Active := L_Gateway_Gas_Alarm_Active,
    VI_Fire_Alarm_Active := L_Gateway_Fire_Alarm_Active,
    VI_Methane_Concentration := GVL_STATE.G_Methane_Sensors[1],
    VI_Lighting_Base_Levels := VIO_Lighting_Base_Levels,
    VI_Socket_States := GVL_STATE.G_Socket_States,
    VI_Blinds_Positions := GVL_STATE.G_Blinds_Positions,
    VI_Active_Scenario := GVL_STATUS.G_Current_Scenario,
    VI_Send_2FA_Req := GVL_COMMAND.G_Send_2FA_Req,
    VI_2FA_Code := GVL_COMMAND.G_2FA_Code_Out,
    VI_Allowed_IPs := GVL_CONFIG.G_Allowed_IPs,
    VO_Telegram_Msg => GVL_GATEWAY.G_Gateway_Telegram_Msg,
    VO_Send_Telegram => GVL_GATEWAY.G_Gateway_Send_Telegram,
    VO_HMI_Status_Message => GVL_GATEWAY.G_Gateway_HMI_Status_Message,
    VO_Data_Ready => GVL_GATEWAY.G_Gateway_Data_Ready,
    VO_Modbus_Registers => GVL_GATEWAY.G_Gateway_Modbus_Registers,
    VO_Arm_Req => GVL_COMMAND.G_Arm_Req,
    VO_Disarm_Req => GVL_COMMAND.G_Disarm_Req,
    VO_PIN_Code => GVL_COMMAND.G_PIN_Code,
    VO_RFID_Tag => GVL_COMMAND.G_RFID_Tag,
    VO_2FA_Code_In => GVL_COMMAND.G_2FA_Code_In,
    VO_Lighting_Override => GVL_COMMAND.G_Lighting_Override,
    VO_Blinds_Override => GVL_COMMAND.G_Blinds_Override,
    VO_Socket_Override => GVL_COMMAND.G_Socket_Override,
    VO_Reset_Errors_Req => GVL_COMMAND.G_Reset_Errors
);

GVL_INTENT_USER.I_Source_Valid := TRUE;
GVL_INTENT_USER.I_Last_Update_MS := VI_System_Time_MS;
GVL_INTENT_USER.I_Arm_Request := GVL_COMMAND.G_Arm_Req;
GVL_INTENT_USER.I_Disarm_Request := GVL_COMMAND.G_Disarm_Req;
GVL_INTENT_USER.I_PIN_Code := GVL_COMMAND.G_PIN_Code;
GVL_INTENT_USER.I_RFID_Tag := GVL_COMMAND.G_RFID_Tag;
GVL_INTENT_USER.I_2FA_Code_In := GVL_COMMAND.G_2FA_Code_In;
GVL_INTENT_USER.I_Lighting_Override_32 := GVL_COMMAND.G_Lighting_Override;
GVL_INTENT_USER.I_Blinds_Override_32 := GVL_COMMAND.G_Blinds_Override;
GVL_INTENT_USER.I_Socket_Override_32 := GVL_COMMAND.G_Socket_Override;
GVL_INTENT_USER.I_Reset_Errors := GVL_COMMAND.G_Reset_Errors;
GVL_INTENT_USER.I_Set_Temp_Req := fbGateway.VO_Set_Temp_Req;
GVL_INTENT_USER.I_Target_Zone := fbGateway.VO_Target_Zone;
GVL_INTENT_USER.I_Target_Temperature := fbGateway.VO_Target_Temp;
GVL_INTENT_USER.I_Set_Vent_Req := fbGateway.VO_Set_Vent_Req;
GVL_INTENT_USER.I_Target_Vent_Speed := fbGateway.VO_Target_Vent_Speed;
GVL_INTENT_USER.I_Set_Config_Req := fbGateway.VO_Set_Config_Req;
GVL_INTENT_USER.I_Time_Sync_Req := fbGateway.VO_Sync_Time_Req;
GVL_INTENT_USER.I_New_Time_MS := fbGateway.VO_New_Time_MS;

// >>> BULK_SYNC_ANCHOR: FB_System_Gateway_Intent <<<
END_FUNCTION_BLOCK

(* ---- FB_System_Health_Orchestrator.st ---- *)
// ==============================================================================
// System health orchestrator helper
//
// Internal helper for PRG_System.
// Owns safety latch update, watchdog, system health aggregation,
// system mode calculation, HMI/fault publication, diagnostic exports,
// and human-readable mode/cause text projection.
// ==============================================================================
FUNCTION_BLOCK FB_System_Health_Orchestrator
VAR_OUTPUT
    VO_First_Fault_Active : BOOL;
    VO_First_Fault_Type : INT;
    VO_First_Fault_Source : INT;
    VO_System_Severity : E_System_Severity;
    VO_Root_Cause : E_System_Root_Cause;
    VO_Watchdog_Fault : BOOL;
END_VAR

VAR
    fbSafety : FB_Safety_Manager;
    fbWatchdog : FB_Watchdog;
    fbSystemHealth : FB_System_Health;
    fbStateManager : FB_State_Manager;
    fbHMIInterface : FB_HMI_Interface;
    fbFaultLogger : FB_Fault_Logger;
END_VAR

fbSafety(
    VI_Gas_Alarm := GVL_HEALTH_BRIDGE.G_Gas_Detected OR GVL_HEALTH_BRIDGE.G_CO_Alarm_Level,
    VI_Leak_Alarm := GVL_HEALTH_BRIDGE.G_Leak_Detected,
    VI_Smoke_Alarm := GVL_HEALTH_BRIDGE.G_Smoke_Detected,
    VI_Reset := GVL_COMMAND.G_Reset_Errors,
    VO_Gas_Latched => GVL_STATE.G_Safety_Gas_Latched,
    VO_Leak_Latched => GVL_STATE.G_Safety_Leak_Latched,
    VO_Smoke_Latched => GVL_STATE.G_Safety_Smoke_Latched,
    VO_Emergency_Stop => GVL_STATE.G_Safety_Emergency_Stop
);

GVL_STATE.G_Freeze_Hardware_Degraded := GVL_STATUS.G_Diagnostics.Backup_Pump_Fault OR GVL_STATUS.G_Diagnostics.Electric_Heater_Fault;
GVL_STATE.G_Freeze_Hardware_Failed := GVL_STATUS.G_Diagnostics.Backup_Pump_Fault AND GVL_STATUS.G_Diagnostics.Electric_Heater_Fault;

fbWatchdog(
    VI_System_Time_MS := GVL_STATUS.G_System_Time_MS
);

fbSystemHealth(
    VI_Smoke_Detected := GVL_HEALTH_BRIDGE.G_Smoke_Detected OR GVL_STATE.G_Safety_Smoke_Latched,
    VI_Gas_Detected := GVL_HEALTH_BRIDGE.G_Gas_Detected OR GVL_STATE.G_Safety_Gas_Latched,
    VI_CO_Warning_Level := GVL_HEALTH_BRIDGE.G_CO_Warning_Level,
    VI_CO_Alarm_Level := GVL_HEALTH_BRIDGE.G_CO_Alarm_Level,
    VI_Leak_Detected := GVL_HEALTH_BRIDGE.G_Leak_Detected OR GVL_STATE.G_Safety_Leak_Latched,
    VI_Sensor_Fault := GVL_STATE.G_Heating_Sensor_Fault OR GVL_STATE.G_DHW_Sensor_Fault OR GVL_STATUS.G_Diagnostics.Manifold_Pressure_Fault_Active OR GVL_STATUS.G_Diagnostics.Manifold_Current_Fault_Active OR GVL_STATUS.G_Diagnostics.Manifold_Return_Temp_Fault_Active,
    VI_IO_Offline := GVL_STATE.G_Heating_IO_Fault OR GVL_STATE.G_DHW_IO_Fault OR GVL_STATE.G_Ventilation_IO_Fault OR GVL_STATE.G_Lighting_IO_Fault,
    VI_Comm_Fault := GVL_STATE.G_Access_Comm_Fault,
    VI_Watchdog_Fault := fbWatchdog.VO_Watchdog_Fault,
    VI_Subsystem_Fault := GVL_STATE.G_Heating_Subsystem_Degraded OR GVL_STATE.G_DHW_Subsystem_Degraded OR GVL_STATE.G_Ventilation_Subsystem_Degraded OR GVL_STATUS.G_Diagnostics.Manifold_Pressure_Fault_Active OR GVL_STATUS.G_Diagnostics.Manifold_Current_Fault_Active OR GVL_STATUS.G_Diagnostics.Manifold_Return_Temp_Fault_Active
);

fbStateManager(
    VI_System_Severity := fbSystemHealth.VO_System_Severity,
    VI_Root_Cause := fbSystemHealth.VO_Root_Cause,
    VI_Freeze_Risk := GVL_STATE.G_Safety_Freeze_Risk
);

fbHMIInterface(
    VI_Severity := fbSystemHealth.VO_System_Severity,
    VI_RootCause := fbSystemHealth.VO_Root_Cause,
    VI_Status_Msg := fbStateManager.VO_Status_Msg
);

fbFaultLogger(
    VI_Severity := fbSystemHealth.VO_System_Severity,
    VI_RootCause := fbSystemHealth.VO_Root_Cause,
    VI_Time_MS := GVL_STATUS.G_System_Time_MS
);

GVL_STATUS.G_System_Mode_Msg := fbStateManager.VO_Status_Msg;

GVL_STATUS.G_Diagnostics.Sensor_Fault :=
    GVL_STATE.G_Heating_Sensor_Fault OR
    GVL_STATE.G_DHW_Sensor_Fault OR
    GVL_STATUS.G_Diagnostics.Manifold_Pressure_Fault_Active OR
    GVL_STATUS.G_Diagnostics.Manifold_Current_Fault_Active OR
    GVL_STATUS.G_Diagnostics.Manifold_Return_Temp_Fault_Active;

GVL_STATUS.G_Diagnostics.IO_Offline :=
    GVL_STATE.G_Heating_IO_Fault OR
    GVL_STATE.G_DHW_IO_Fault OR
    GVL_STATE.G_Ventilation_IO_Fault OR
    GVL_STATE.G_Lighting_IO_Fault;

GVL_STATUS.G_Diagnostics.Subsystem_Degraded :=
    GVL_STATE.G_Heating_Subsystem_Degraded OR
    GVL_STATE.G_DHW_Subsystem_Degraded OR
    GVL_STATE.G_Ventilation_Subsystem_Degraded OR
    GVL_STATUS.G_Diagnostics.Manifold_Pressure_Fault_Active OR
    GVL_STATUS.G_Diagnostics.Manifold_Current_Fault_Active OR
    GVL_STATUS.G_Diagnostics.Manifold_Return_Temp_Fault_Active;

GVL_GATEWAY.G_Gateway_HMI_Status_Message := fbHMIInterface.VO_HMI_Status_Text;
IF fbFaultLogger.VO_Last_Event_Text <> '' THEN
    GVL_HEALTH_BRIDGE.G_Last_Fault_Event_Text := fbFaultLogger.VO_Last_Event_Text;
END_IF;

GVL_STATE.G_System_Mode := fbStateManager.VO_System_Mode;

CASE GVL_STATE.G_System_Mode OF
    E_System_Operating_Mode.MODE_SAFE_STOP:
        GVL_STATE.G_System_Mode_Text := 'SAFE_STOP';

    E_System_Operating_Mode.MODE_FREEZE_PROTECTION:
        GVL_STATE.G_System_Mode_Text := 'FREEZE_PROTECTION';

    E_System_Operating_Mode.MODE_DEGRADED:
        GVL_STATE.G_System_Mode_Text := 'DEGRADED';

    ELSE
        GVL_STATE.G_System_Mode_Text := 'NORMAL';
END_CASE;

CASE fbSystemHealth.VO_Root_Cause OF
    E_System_Root_Cause.ROOT_FIRE:
        GVL_STATUS.G_System_Mode_Cause := 'Пожар/дым';
    E_System_Root_Cause.ROOT_GAS_LEAK:
        GVL_STATUS.G_System_Mode_Cause := 'Утечка газа';
    E_System_Root_Cause.ROOT_CO_CRITICAL:
        GVL_STATUS.G_System_Mode_Cause := 'Критический CO';
    E_System_Root_Cause.ROOT_CO_WARNING:
        GVL_STATUS.G_System_Mode_Cause := 'Повышенный CO';
    E_System_Root_Cause.ROOT_WATER_LEAK:
        GVL_STATUS.G_System_Mode_Cause := 'Протечка воды';
    E_System_Root_Cause.ROOT_WATCHDOG_FAULT:
        GVL_STATUS.G_System_Mode_Cause := 'Ошибка watchdog';
    E_System_Root_Cause.ROOT_IO_OFFLINE:
        GVL_STATUS.G_System_Mode_Cause := 'Недоступен модуль IO';
    E_System_Root_Cause.ROOT_COMM_FAULT:
        GVL_STATUS.G_System_Mode_Cause := 'Ошибка связи';
    E_System_Root_Cause.ROOT_SENSOR_FAULT:
        GVL_STATUS.G_System_Mode_Cause := 'Ошибка датчика';
    E_System_Root_Cause.ROOT_SUBSYSTEM_FAULT:
        GVL_STATUS.G_System_Mode_Cause := 'Ошибка подсистемы';
    ELSE
        GVL_STATUS.G_System_Mode_Cause := 'Аварийные режимы отсутствуют';
END_CASE;

VO_First_Fault_Active := fbSystemHealth.VO_First_Fault_Active;
VO_First_Fault_Type := fbSystemHealth.VO_First_Fault_Type;
VO_First_Fault_Source := fbSystemHealth.VO_First_Fault_Source;
VO_System_Severity := fbSystemHealth.VO_System_Severity;
VO_Root_Cause := fbSystemHealth.VO_Root_Cause;
VO_Watchdog_Fault := fbWatchdog.VO_Watchdog_Fault;

GVL_STATUS.G_System_Mode_Msg := fbStateManager.VO_Status_Msg;

// >>> BULK_SYNC_ANCHOR: FB_System_Health_Orchestrator <<<
END_FUNCTION_BLOCK

(* ---- FB_Water_Isolation_Authority_Arbitrator.st ---- *)
FUNCTION_BLOCK FB_Water_Isolation_Authority_Arbitrator
VAR_INPUT
    VI_Enable : BOOL;
    VI_System_Time_MS : UDINT;
END_VAR
VAR
    L_i : INT;
    L_Runtime : ST_Water_Isolation_Runtime_State;
    L_Traversal : ST_Water_Graph_Traversal_State;
    L_Authority : ST_Water_Isolation_Authority_State;
    L_Empty_Authority : ST_Water_Isolation_Authority_State;
    L_Any_Selective : BOOL;
    L_Any_Global : BOOL;
    L_Any_Denied : BOOL;
END_VAR

IF NOT VI_Enable THEN
    GVL_Water_Isolation_Authority.G_Authority_Valid := FALSE;
    RETURN;
END_IF;

L_Any_Selective := FALSE;
L_Any_Global := FALSE;
L_Any_Denied := FALSE;

FOR L_i := 1 TO GVL_CONSTANTS.C_MAX_FLOOD_SENSORS DO

    L_Runtime := GVL_Water_Isolation_Runtime.G_Isolation_Runtime_State[L_i];
    L_Traversal := GVL_Water_Orchestration.G_Traversal_State[L_i];

    L_Authority := L_Empty_Authority;
    L_Authority.Decision_Valid := TRUE;
    L_Authority.Decision_System_Time_MS := VI_System_Time_MS;

    L_Authority.Isolation_Requested := L_Runtime.Isolation_Requested;
    L_Authority.Selective_Candidate := L_Runtime.Selective_Isolation_Requested;
    L_Authority.Global_Fallback_Candidate := L_Runtime.Global_Isolation_Requested;

    L_Authority.Hydraulic_Zone_Id := L_Runtime.Hydraulic_Zone_Id;
    L_Authority.Isolation_Group_Id := L_Runtime.Isolation_Group_Id;
    L_Authority.Valve_Group_Id := L_Runtime.Valve_Group_Id;

    // Orchestration-derived authority.
    L_Authority.Mapping_Valid := L_Traversal.Traversal_Valid;

    L_Authority.Deterministic_Target_Valid :=
        (L_Runtime.Valve_Group_Id <> 0)
        AND NOT L_Traversal.Traversal_Conflict
        AND NOT L_Traversal.Traversal_Ambiguous;

    L_Authority.Safety_Context_Allows_Selective :=
        NOT GVL_INTENT_SAFETY.I_Water_Main_Close_Required;

    IF NOT L_Authority.Isolation_Requested THEN

        L_Authority.Decision_Code := 0;
        L_Authority.Decision_Text := 'No authority required';

    ELSIF NOT L_Authority.Mapping_Valid
       OR NOT L_Authority.Deterministic_Target_Valid
       OR NOT L_Authority.Safety_Context_Allows_Selective THEN

        L_Authority.Global_Fallback_Required := TRUE;
        L_Authority.Authority_Denied := TRUE;

        L_Authority.Decision_Code := 2;
        L_Authority.Decision_Text := 'Global fallback authority active';

    ELSE

        L_Authority.Selective_Authority_Allowed := TRUE;

        L_Authority.Decision_Code := 10;
        L_Authority.Decision_Text := 'Selective authority granted';

    END_IF;

    GVL_Water_Isolation_Authority.G_Authority_State[L_i] :=
        L_Authority;

    L_Any_Selective :=
        L_Any_Selective
        OR L_Authority.Selective_Authority_Allowed;

    L_Any_Global :=
        L_Any_Global
        OR L_Authority.Global_Fallback_Required;

    L_Any_Denied :=
        L_Any_Denied
        OR L_Authority.Authority_Denied;

END_FOR;

GVL_Water_Isolation_Authority.G_Any_Selective_Authority_Allowed :=
    L_Any_Selective;

GVL_Water_Isolation_Authority.G_Any_Global_Fallback_Required :=
    L_Any_Global;

GVL_Water_Isolation_Authority.G_Any_Authority_Denied :=
    L_Any_Denied;

GVL_Water_Isolation_Authority.G_Authority_Valid := TRUE;
GVL_Water_Isolation_Authority.G_Last_Update_MS := VI_System_Time_MS;

IF L_Any_Global THEN
    GVL_Water_Isolation_Authority.G_Status_Code := 2;
    GVL_Water_Isolation_Authority.G_Status_Text :=
        'Global fallback authority active';
ELSIF L_Any_Selective THEN
    GVL_Water_Isolation_Authority.G_Status_Code := 1;
    GVL_Water_Isolation_Authority.G_Status_Text :=
        'Selective orchestration authority active';
ELSE
    GVL_Water_Isolation_Authority.G_Status_Code := 0;
    GVL_Water_Isolation_Authority.G_Status_Text :=
        'Authority arbitration healthy';
END_IF;

END_FUNCTION_BLOCK

(* ---- FB_Water_Isolation_Path_Resolver.st ---- *)
FUNCTION_BLOCK FB_Water_Isolation_Path_Resolver
VAR_INPUT
    VI_Enable : BOOL;
    VI_System_Time_MS : UDINT;
END_VAR
VAR
    L_i : INT;

    L_Edge : ST_Water_Hydraulic_Topology_Edge;
    L_Path : ST_Water_Isolation_Path_Runtime_State;
    L_Validation : ST_Water_Topology_Validation_State;

    L_Empty_Edge : ST_Water_Hydraulic_Topology_Edge;
    L_Empty_Path : ST_Water_Isolation_Path_Runtime_State;

    L_Any_Shared_Trunk : BOOL;
    L_Any_Conflict : BOOL;
    L_Any_Fallback : BOOL;
END_VAR

IF NOT VI_Enable THEN
    GVL_Water_Hydraulic_Graph.G_Runtime_Valid := FALSE;
    RETURN;
END_IF;

L_Any_Shared_Trunk := FALSE;
L_Any_Conflict := FALSE;
L_Any_Fallback := FALSE;

FOR L_i := 1 TO GVL_CONSTANTS.C_MAX_FLOOD_SENSORS DO

    L_Validation :=
        GVL_Water_Topology_Validation.G_Validation_State[L_i];

    // Graph edge publication.
    L_Edge := L_Empty_Edge;
    L_Edge.Runtime_Valid := TRUE;

    L_Edge.Edge_Id := TO_UINT(L_i);

    L_Edge.Upstream_Segment_Id :=
        GVL_Water_Hydraulic_Topology.G_Topology_Node[L_i].Hydraulic_Segment_Id;

    L_Edge.Downstream_Segment_Id :=
        GVL_Water_Hydraulic_Topology.G_Topology_Node[L_i].Hydraulic_Zone_Id;

    L_Edge.Isolation_Group_Id :=
        GVL_Water_Hydraulic_Topology.G_Topology_Node[L_i].Isolation_Group_Id;

    L_Edge.Valve_Group_Id :=
        GVL_Water_Hydraulic_Topology.G_Topology_Node[L_i].Valve_Group_Id;

    // Shared trunk semantics.
    IF L_Edge.Valve_Group_Id = 3 THEN
        L_Edge.Shared_Trunk := TRUE;
        L_Edge.Cross_Zone_Dependency := TRUE;
    END_IF;

    L_Edge.Dependency_Valid :=
        L_Validation.Topology_Valid;

    L_Edge.Dependency_Ambiguous :=
        L_Validation.Topology_Ambiguous;

    L_Edge.Selective_Isolation_Allowed :=
        L_Validation.Selective_Isolation_Allowed;

    L_Edge.Global_Fallback_Required :=
        L_Validation.Global_Fallback_Required;

    // Isolation path runtime.
    L_Path := L_Empty_Path;
    L_Path.Runtime_Valid := TRUE;

    L_Path.Runtime_System_Time_MS :=
        VI_System_Time_MS;

    L_Path.Sensor_Id := TO_UINT(L_i);

    L_Path.Isolation_Path_Valid :=
        L_Edge.Dependency_Valid;

    L_Path.Isolation_Path_Ambiguous :=
        L_Edge.Dependency_Ambiguous;

    L_Path.Active_Isolation_Group_Id :=
        L_Edge.Isolation_Group_Id;

    L_Path.Active_Valve_Group_Id :=
        L_Edge.Valve_Group_Id;

    L_Path.Shared_Trunk_Impact :=
        L_Edge.Shared_Trunk;

    L_Path.Cross_Zone_Impact :=
        L_Edge.Cross_Zone_Dependency;

    L_Path.Selective_Isolation_Allowed :=
        L_Edge.Selective_Isolation_Allowed;

    L_Path.Global_Fallback_Required :=
        L_Edge.Global_Fallback_Required;

    // Multi-valve/shared-trunk path.
    IF L_Path.Shared_Trunk_Impact THEN
        L_Path.Multi_Valve_Path := TRUE;
    END_IF;

    // Conflict detection.
    IF L_Path.Isolation_Path_Ambiguous THEN
        L_Path.Conflict_Detected := TRUE;
    END_IF;

    // Conservative escalation.
    IF L_Path.Conflict_Detected THEN
        L_Path.Global_Fallback_Required := TRUE;
        L_Path.Selective_Isolation_Allowed := FALSE;

        L_Path.Status_Code := 2;
        L_Path.Status_Text :=
            'Isolation path conflict detected';

    ELSIF L_Path.Shared_Trunk_Impact THEN
        L_Path.Status_Code := 1;
        L_Path.Status_Text :=
            'Shared trunk isolation path active';

    ELSE
        L_Path.Status_Code := 0;
        L_Path.Status_Text :=
            'Isolation path resolved';
    END_IF;

    GVL_Water_Hydraulic_Graph.G_Topology_Edge[L_i] :=
        L_Edge;

    GVL_Water_Hydraulic_Graph.G_Isolation_Path[L_i] :=
        L_Path;

    L_Any_Shared_Trunk :=
        L_Any_Shared_Trunk
        OR L_Path.Shared_Trunk_Impact;

    L_Any_Conflict :=
        L_Any_Conflict
        OR L_Path.Conflict_Detected;

    L_Any_Fallback :=
        L_Any_Fallback
        OR L_Path.Global_Fallback_Required;

END_FOR;

GVL_Water_Hydraulic_Graph.G_Any_Shared_Trunk :=
    L_Any_Shared_Trunk;

GVL_Water_Hydraulic_Graph.G_Any_Conflict :=
    L_Any_Conflict;

GVL_Water_Hydraulic_Graph.G_Any_Global_Fallback_Required :=
    L_Any_Fallback;

GVL_Water_Hydraulic_Graph.G_Runtime_Valid := TRUE;
GVL_Water_Hydraulic_Graph.G_Last_Update_MS := VI_System_Time_MS;

IF L_Any_Conflict THEN
    GVL_Water_Hydraulic_Graph.G_Status_Code := 2;
    GVL_Water_Hydraulic_Graph.G_Status_Text :=
        'Hydraulic graph conflicts detected';
ELSIF L_Any_Shared_Trunk THEN
    GVL_Water_Hydraulic_Graph.G_Status_Code := 1;
    GVL_Water_Hydraulic_Graph.G_Status_Text :=
        'Shared trunk governance active';
ELSE
    GVL_Water_Hydraulic_Graph.G_Status_Code := 0;
    GVL_Water_Hydraulic_Graph.G_Status_Text :=
        'Hydraulic graph runtime healthy';
END_IF;

END_FUNCTION_BLOCK

(* ---- FB_Water_Leakage_Manager.st ---- *)
FUNCTION_BLOCK FB_Water_Leakage_Manager
VAR_INPUT
    VI_System_Time_MS : UDINT;
    VI_IsActivePLC    : BOOL;
    VI_Config         : ST_Flood_Global_Config;
END_VAR

VAR_IN_OUT
    VI_Sensors : ARRAY[1..GVL_CONSTANTS.C_MAX_FLOOD_SENSORS] OF BOOL;
END_VAR

VAR_OUTPUT
    VO_Status_Msg     : STRING(200);
    VO_Leak_Detected      : BOOL;
    VO_Leak_Warning_Level : BOOL;
END_VAR

VAR
    L_i             : INT;
    L_Sensor_Timers : ARRAY[1..GVL_CONSTANTS.C_MAX_FLOOD_SENSORS] OF FB_System_Timer;
    L_Any_Leak      : BOOL;
    L_Any_Warning   : BOOL;
END_VAR

IF NOT VI_IsActivePLC THEN RETURN; END_IF;

L_Any_Leak := FALSE;
L_Any_Warning := FALSE;

FOR L_i := 1 TO GVL_CONSTANTS.C_MAX_FLOOD_SENSORS DO
    L_Sensor_Timers[L_i](
        IN := VI_Sensors[L_i],
        PT := TO_TIME(VI_Config.min_duration_ms + VI_Config.warning_duration_ms),
        VI_System_Time_MS := VI_System_Time_MS
    );

    IF L_Sensor_Timers[L_i].ET >= TO_TIME(VI_Config.min_duration_ms) THEN
        L_Any_Warning := TRUE;

        IF L_Sensor_Timers[L_i].Q THEN
            L_Any_Leak := TRUE;
        END_IF;
    END_IF;
END_FOR;

// Manual latch instead of RS
IF GVL_INTENT_USER.I_Reset_Errors THEN
    VO_Leak_Detected := FALSE;
ELSIF L_Any_Leak THEN
    VO_Leak_Detected := TRUE;
END_IF;

VO_Leak_Warning_Level := L_Any_Warning;

IF VO_Leak_Detected THEN
    VO_Status_Msg := 'АВАРИЯ: ПРОТЕЧКА ВОДЫ.';
ELSIF L_Any_Warning THEN
    VO_Status_Msg := 'ПРЕДУПРЕЖДЕНИЕ: ОБНАРУЖЕНА ВОДА.';
ELSE
    VO_Status_Msg := 'Система контроля протечек в норме';
END_IF;
// >>> BULK_SYNC_ANCHOR: FB_Water_Leakage_Manager <<<
END_FUNCTION_BLOCK

(* ---- FB_Water_Orchestration_Runtime.st ---- *)
FUNCTION_BLOCK FB_Water_Orchestration_Runtime
VAR_INPUT
    VI_Enable : BOOL;
    VI_System_Time_MS : UDINT;
END_VAR
VAR
    L_i : INT;

    L_Path : ST_Water_Isolation_Path_Runtime_State;
    L_Traversal : ST_Water_Graph_Traversal_State;
    L_Orchestration : ST_Water_Orchestration_Runtime_State;

    L_Empty_Traversal : ST_Water_Graph_Traversal_State;
    L_Empty_Orchestration : ST_Water_Orchestration_Runtime_State;

    L_Any_Conflict : BOOL;
    L_Any_Escalation : BOOL;
END_VAR

IF NOT VI_Enable THEN
    GVL_Water_Orchestration.G_Runtime_Valid := FALSE;
    RETURN;
END_IF;

L_Any_Conflict := FALSE;
L_Any_Escalation := FALSE;

FOR L_i := 1 TO GVL_CONSTANTS.C_MAX_FLOOD_SENSORS DO

    L_Path :=
        GVL_Water_Hydraulic_Graph.G_Isolation_Path[L_i];

    // Traversal runtime.
    L_Traversal := L_Empty_Traversal;
    L_Traversal.Runtime_Valid := TRUE;

    L_Traversal.Runtime_System_Time_MS :=
        VI_System_Time_MS;

    L_Traversal.Sensor_Id := TO_UINT(L_i);

    L_Traversal.Start_Segment_Id :=
        L_Path.Active_Isolation_Group_Id;

    L_Traversal.Target_Valve_Group_Id :=
        L_Path.Active_Valve_Group_Id;

    L_Traversal.Shared_Trunk_Traversal :=
        L_Path.Shared_Trunk_Impact;

    L_Traversal.Upstream_Dependency_Detected :=
        L_Path.Shared_Trunk_Impact;

    L_Traversal.Downstream_Impact_Detected :=
        L_Path.Cross_Zone_Impact;

    L_Traversal.Traversal_Valid :=
        L_Path.Isolation_Path_Valid;

    L_Traversal.Traversal_Conflict :=
        L_Path.Conflict_Detected;

    L_Traversal.Traversal_Ambiguous :=
        L_Path.Isolation_Path_Ambiguous;

    IF L_Path.Multi_Valve_Path THEN
        L_Traversal.Dependency_Depth := 2;
    ELSE
        L_Traversal.Dependency_Depth := 1;
    END_IF;

    L_Traversal.Selective_Path_Allowed :=
        L_Path.Selective_Isolation_Allowed;

    L_Traversal.Global_Fallback_Required :=
        L_Path.Global_Fallback_Required;

    // Orchestration runtime.
    L_Orchestration := L_Empty_Orchestration;
    L_Orchestration.Runtime_Valid := TRUE;

    L_Orchestration.Runtime_System_Time_MS :=
        VI_System_Time_MS;

    L_Orchestration.Isolation_Sequence_Active :=
        L_Traversal.Traversal_Valid;

    L_Orchestration.Shared_Trunk_Sequencing :=
        L_Traversal.Shared_Trunk_Traversal;

    L_Orchestration.Staged_Close_Required :=
        L_Path.Multi_Valve_Path;

    L_Orchestration.Recovery_Sequence_Active :=
        GVL_INTENT_SAFETY.I_Water_Selective_Recovery_Allowed;

    L_Orchestration.Staged_Open_Required :=
        L_Orchestration.Recovery_Sequence_Active
        AND L_Path.Multi_Valve_Path;

    L_Orchestration.Observation_Window_Active :=
        L_Orchestration.Recovery_Sequence_Active;

    // Conservative sequencing governance.
    IF L_Traversal.Traversal_Conflict
       OR L_Traversal.Traversal_Ambiguous THEN

        L_Orchestration.Rollback_Required := TRUE;
        L_Orchestration.Escalation_Required := TRUE;
        L_Orchestration.Sequencing_Valid := FALSE;

        L_Orchestration.Status_Code := 2;
        L_Orchestration.Status_Text :=
            'Orchestration conflict escalation active';

    ELSE

        L_Orchestration.Sequencing_Valid := TRUE;

        IF L_Orchestration.Shared_Trunk_Sequencing THEN
            L_Orchestration.Status_Code := 1;
            L_Orchestration.Status_Text :=
                'Shared trunk orchestration active';
        ELSE
            L_Orchestration.Status_Code := 0;
            L_Orchestration.Status_Text :=
                'Deterministic orchestration active';
        END_IF;

    END_IF;

    GVL_Water_Orchestration.G_Traversal_State[L_i] :=
        L_Traversal;

    GVL_Water_Orchestration.G_Orchestration_State[L_i] :=
        L_Orchestration;

    L_Any_Conflict :=
        L_Any_Conflict
        OR L_Traversal.Traversal_Conflict;

    L_Any_Escalation :=
        L_Any_Escalation
        OR L_Orchestration.Escalation_Required;

END_FOR;

GVL_Water_Orchestration.G_Topology_Version := 1;
GVL_Water_Orchestration.G_Config_Runtime_Ready := TRUE;

GVL_Water_Orchestration.G_Any_Traversal_Conflict :=
    L_Any_Conflict;

GVL_Water_Orchestration.G_Any_Escalation_Required :=
    L_Any_Escalation;

GVL_Water_Orchestration.G_Runtime_Valid := TRUE;
GVL_Water_Orchestration.G_Last_Update_MS := VI_System_Time_MS;

IF L_Any_Escalation THEN
    GVL_Water_Orchestration.G_Status_Code := 2;
    GVL_Water_Orchestration.G_Status_Text :=
        'Water orchestration escalation active';
ELSIF L_Any_Conflict THEN
    GVL_Water_Orchestration.G_Status_Code := 1;
    GVL_Water_Orchestration.G_Status_Text :=
        'Water orchestration conflict detected';
ELSE
    GVL_Water_Orchestration.G_Status_Code := 0;
    GVL_Water_Orchestration.G_Status_Text :=
        'Water orchestration runtime healthy';
END_IF;

END_FUNCTION_BLOCK

(* ---- FB_Water_Recovery_Runtime.st ---- *)
FUNCTION_BLOCK FB_Water_Recovery_Runtime
VAR_INPUT
    VI_Enable : BOOL;
    VI_System_Time_MS : UDINT;
END_VAR
VAR
    L_i : INT;
    L_Feedback : ST_Water_Valve_Feedback_State;
    L_State : ST_Water_Recovery_Runtime_State;
    L_Any_Denied : BOOL;
    L_Any_Unsafe : BOOL;
END_VAR

IF NOT VI_Enable THEN
    GVL_Water_Recovery_Runtime.G_Runtime_Valid := FALSE;
    RETURN;
END_IF;

FOR L_i := 1 TO GVL_CONSTANTS.C_MAX_FLOOD_SENSORS DO
    L_Feedback := GVL_Water_Valve_Feedback.G_Valve_Feedback_State[L_i];

    L_State.Runtime_Valid := TRUE;
    L_State.Runtime_System_Time_MS := VI_System_Time_MS;
    L_State.Recovery_Requested := GVL_INTENT_SAFETY.I_Water_Selective_Recovery_Allowed;
    L_State.Valve_Degraded := L_Feedback.Valve_Degraded;
    L_State.Confirmation_Healthy := NOT L_Feedback.Feedback_Conflict;
    L_State.Recovery_Target_Valid := L_Feedback.Valve_Group_Id <> 0;

    IF NOT L_State.Recovery_Target_Valid THEN
        L_State.Recovery_Denied := TRUE;
        L_State.Status_Code := 1;
        L_State.Status_Text := 'Recovery target invalid';
    ELSIF L_State.Valve_Degraded THEN
        L_State.Recovery_Denied := TRUE;
        L_State.Unsafe_Recovery_Detected := TRUE;
        L_State.Status_Code := 2;
        L_State.Status_Text := 'Recovery blocked by valve state';
    ELSIF NOT L_State.Confirmation_Healthy THEN
        L_State.Recovery_Denied := TRUE;
        L_State.Status_Code := 3;
        L_State.Status_Text := 'Recovery blocked by confirmation state';
    ELSE
        L_State.Recovery_Allowed := TRUE;
        L_State.Observation_Window_Active := TRUE;
        L_State.Status_Code := 0;
        L_State.Status_Text := 'Recovery governance healthy';
    END_IF;

    GVL_Water_Recovery_Runtime.G_Recovery_State[L_i] := L_State;
    L_Any_Denied := L_Any_Denied OR L_State.Recovery_Denied;
    L_Any_Unsafe := L_Any_Unsafe OR L_State.Unsafe_Recovery_Detected;
END_FOR;

GVL_Water_Recovery_Runtime.G_Any_Recovery_Denied := L_Any_Denied;
GVL_Water_Recovery_Runtime.G_Any_Unsafe_Recovery := L_Any_Unsafe;
GVL_Water_Recovery_Runtime.G_Runtime_Valid := TRUE;
GVL_Water_Recovery_Runtime.G_Last_Update_MS := VI_System_Time_MS;

IF L_Any_Unsafe THEN
    GVL_Water_Recovery_Runtime.G_Status_Code := 2;
    GVL_Water_Recovery_Runtime.G_Status_Text := 'Recovery risk detected';
ELSIF L_Any_Denied THEN
    GVL_Water_Recovery_Runtime.G_Status_Code := 1;
    GVL_Water_Recovery_Runtime.G_Status_Text := 'Recovery governance denied';
ELSE
    GVL_Water_Recovery_Runtime.G_Status_Code := 0;
    GVL_Water_Recovery_Runtime.G_Status_Text := 'Recovery governance healthy';
END_IF;

END_FUNCTION_BLOCK
